LIN {X 0,Y 582.697,Z 999.252,A -85,B 0,C 180,E1 27417.863,E2 27417.863} C_VEL
LIN {X 0,Y 579.637,Z 1018.476,A -85,B 0,C 180,E1 27415.72,E2 27415.72} C_VEL
LIN {X 0,Y 576.832,Z 1036.876,A -85,B 0,C 180,E1 27413.377,E2 27413.377} C_VEL
LIN {X 0,Y 574.399,Z 1053.777,A -85,B 0,C 180,E1 27410.931,E2 27410.931} C_VEL
LIN {X 0,Y 572.425,Z 1069.156,A -85,B 0,C 180,E1 27408.385,E2 27408.385} C_VEL
LIN {X 0,Y 570.966,Z 1081.996,A -85,B 0,C 180,E1 27405.955,E2 27405.955} C_VEL
LIN {X 0,Y 569.794,Z 1094.009,A -85,B 0,C 180,E1 27403.325,E2 27403.325} C_VEL
LIN {X 0,Y 568.899,Z 1104.701,A -85,B 0,C 180,E1 27400.565,E2 27400.565} C_VEL
LIN {X 0,Y 568.443,Z 1112.638,A -85,B 0,C 180,E1 27398.127,E2 27398.127} C_VEL
LIN {X 0,Y 568.122,Z 1119.365,A -85,B 0,C 180,E1 27395.6,E2 27395.6} C_VEL
LIN {X 0,Y 567.953,Z 1124.698,A -85,B 0,C 180,E1 27393.071,E2 27393.071} C_VEL
LIN {X 0,Y 567.932,Z 1128.442,A -85,B 0,C 180,E1 27390.581,E2 27390.581} C_VEL
LIN {X 0,Y 567.917,Z 1130.903,A -85,B 0,C 180,E1 27388.04,E2 27388.04} C_VEL
LIN {X 0,Y 567.902,Z 1131.896,A -85,B 0,C 180,E1 27385.554,E2 27385.554} C_VEL
LIN {X 0,Y 567.866,Z 1131.496,A -85,B 0,C 180,E1 27382.901,E2 27382.901} C_VEL
LIN {X 0,Y 567.918,Z 1129.69,A -85,B 0,C 180,E1 27380.402,E2 27380.402} C_VEL
LIN {X 0,Y 567.966,Z 1126.174,A -85,B 0,C 180,E1 27377.732,E2 27377.732} C_VEL
LIN {X 0,Y 568.103,Z 1120.964,A -85,B 0,C 180,E1 27374.995,E2 27374.995} C_VEL
LIN {X 0,Y 568.345,Z 1114.143,A -85,B 0,C 180,E1 27372.291,E2 27372.291} C_VEL
LIN {X 0,Y 568.803,Z 1106.34,A -85,B 0,C 180,E1 27369.818,E2 27369.818} C_VEL
LIN {X 0,Y 569.536,Z 1096.854,A -85,B 0,C 180,E1 27367.262,E2 27367.262} C_VEL
LIN {X 0,Y 570.678,Z 1084.618,A -85,B 0,C 180,E1 27364.488,E2 27364.488} C_VEL
LIN {X 0,Y 572.097,Z 1071.819,A -85,B 0,C 180,E1 27362.003,E2 27362.003} C_VEL
LIN {X 0,Y 573.974,Z 1057.101,A -85,B 0,C 180,E1 27359.501,E2 27359.501} C_VEL
LIN {X 0,Y 576.32,Z 1040.394,A -85,B 0,C 180,E1 27357.016,E2 27357.016} C_VEL
LIN {X 0,Y 578.934,Z 1023.074,A -85,B 0,C 180,E1 27354.748,E2 27354.748} C_VEL
LIN {X 0,Y 582,Z 1003.502,A -85,B 0,C 180,E1 27352.497,E2 27352.497} C_VEL
LIN {X 0,Y 585.241,Z 983.342,A -85,B 0,C 180,E1 27350.461,E2 27350.461} C_VEL
LIN {X 0,Y 588.632,Z 962.34,A -85,B 0,C 180,E1 27348.586,E2 27348.586} C_VEL
LIN {X 0,Y 592.216,Z 939.835,A -85,B 0,C 180,E1 27346.825,E2 27346.825} C_VEL
LIN {X 0,Y 595.837,Z 916.143,A -85,B 0,C 180,E1 27345.222,E2 27345.222} C_VEL
LIN {X 0,Y 599.193,Z 893.145,A -85,B 0,C 180,E1 27343.868,E2 27343.868} C_VEL
LIN {X 0,Y 602.06,Z 871.003,A -85,B 0,C 180,E1 27342.755,E2 27342.755} C_VEL
LIN {X 0,Y 604.46,Z 849.4,A -85,B 0,C 180,E1 27341.831,E2 27341.831} C_VEL
LIN {X 0,Y 606.973,Z 822.591,A -85,B 0,C 180,E1 27340.888,E2 27340.888} C_VEL
LIN {X 0,Y 608.639,Z 799.863,A -85,B 0,C 180,E1 27340.257,E2 27340.257} C_VEL
LIN {X 0,Y 609.845,Z 778.887,A -85,B 0,C 180,E1 27339.791,E2 27339.791} C_VEL
LIN {X 0,Y 610.75,Z 757.121,A -85,B 0,C 180,E1 27339.422,E2 27339.422} C_VEL
LIN {X 0,Y 615.009,Z 585.018,A -85,B 0,C 180,E1 27337.044,E2 27337.044} C_VEL
LIN {X 0,Y 619.202,Z 468.417,A -85,B 0,C 180,E1 27335.305,E2 27335.305} C_VEL
LIN {X 0,Y 621.386,Z 419.773,A -85,B 0,C 180,E1 27334.516,E2 27334.516} C_VEL
LIN {X 0,Y 613.039,Z 405.628,A -85,B 0,C 180,E1 27332.992,E2 27332.992} C_VEL
LIN {X 0,Y 608.359,Z 397.704,A -85,B 0,C 180,E1 27331.887,E2 27331.887} C_VEL
LIN {X 0,Y 605.73,Z 393.264,A -85,B 0,C 180,E1 27331.075,E2 27331.075} C_VEL
LIN {X 0,Y 603.613,Z 389.51,A -85,B 0,C 180,E1 27330.201,E2 27330.201} C_VEL
LIN {X 0,Y 602.051,Z 387.195,A -85,B 0,C 180,E1 27329.068,E2 27329.068} C_VEL
LIN {X 0,Y 601.397,Z 389.334,A -85,B 0,C 180,E1 27328.306,E2 27328.306} C_VEL
LIN {X 0,Y 601.328,Z 391.857,A -85,B 0,C 180,E1 27327.678,E2 27327.678} C_VEL
LIN {X 0,Y 602.239,Z 397.51,A -85,B 0,C 180,E1 27326.663,E2 27326.663} C_VEL
LIN {X 0,Y 604.241,Z 405.255,A -85,B 0,C 180,E1 27325.619,E2 27325.619} C_VEL
LIN {X 0,Y 608.329,Z 418.436,A -85,B 0,C 180,E1 27324.303,E2 27324.303} C_VEL
LIN {X 0,Y 613.755,Z 430.748,A -85,B 0,C 180,E1 27323.141,E2 27323.141} C_VEL
LIN {X 0,Y 617.349,Z 460.837,A -85,B 0,C 180,E1 27321.984,E2 27321.984} C_VEL
LIN {X 0,Y 619.834,Z 475.835,A -85,B 0,C 180,E1 27321.397,E2 27321.397} C_VEL
LIN {X 0,Y 615.945,Z 588.673,A -85,B 0,C 180,E1 27319.681,E2 27319.681} C_VEL
LIN {X 0,Y 612.665,Z 730.462,A -85,B 0,C 180,E1 27317.702,E2 27317.702} C_VEL
LIN {X 0,Y 609.681,Z 897.665,A -85,B 0,C 180,E1 27315.502,E2 27315.502} C_VEL
LIN {X 0,Y 608.295,Z 927.071,A -85,B 0,C 180,E1 27314.989,E2 27314.989} C_VEL
LIN {X 0,Y 606.632,Z 952.665,A -85,B 0,C 180,E1 27314.385,E2 27314.385} C_VEL
LIN {X 0,Y 605.035,Z 974.265,A -85,B 0,C 180,E1 27313.764,E2 27313.764} C_VEL
LIN {X 0,Y 603.312,Z 995.06,A -85,B 0,C 180,E1 27313.064,E2 27313.064} C_VEL
LIN {X 0,Y 601.59,Z 1014.742,A -85,B 0,C 180,E1 27312.3,E2 27312.3} C_VEL
LIN {X 0,Y 599.545,Z 1035.386,A -85,B 0,C 180,E1 27311.395,E2 27311.395} C_VEL
LIN {X 0,Y 597.906,Z 1050.557,A -85,B 0,C 180,E1 27310.644,E2 27310.644} C_VEL
LIN {X 0,Y 595.718,Z 1066.737,A -85,B 0,C 180,E1 27309.691,E2 27309.691} C_VEL
LIN {X 0,Y 592.722,Z 1086.305,A -85,B 0,C 180,E1 27308.374,E2 27308.374} C_VEL
LIN {X 0,Y 589.851,Z 1104.551,A -85,B 0,C 180,E1 27306.997,E2 27306.997} C_VEL
LIN {X 0,Y 586.954,Z 1122.563,A -85,B 0,C 180,E1 27305.483,E2 27305.483} C_VEL
LIN {X 0,Y 583.573,Z 1143.707,A -85,B 0,C 180,E1 27303.484,E2 27303.484} C_VEL
LIN {X 0,Y 580.57,Z 1162.442,A -85,B 0,C 180,E1 27301.455,E2 27301.455} C_VEL
LIN {X 0,Y 578.226,Z 1177.518,A -85,B 0,C 180,E1 27299.64,E2 27299.64} C_VEL
LIN {X 0,Y 575.845,Z 1193.458,A -85,B 0,C 180,E1 27297.508,E2 27297.508} C_VEL
LIN {X 0,Y 573.558,Z 1210.189,A -85,B 0,C 180,E1 27294.953,E2 27294.953} C_VEL
LIN {X 0,Y 571.964,Z 1222.995,A -85,B 0,C 180,E1 27292.727,E2 27292.727} C_VEL
LIN {X 0,Y 570.657,Z 1234.974,A -85,B 0,C 180,E1 27290.378,E2 27290.378} C_VEL
LIN {X 0,Y 569.454,Z 1247.679,A -85,B 0,C 180,E1 27287.473,E2 27287.473} C_VEL
LIN {X 0,Y 568.84,Z 1256.157,A -85,B 0,C 180,E1 27285.183,E2 27285.183} C_VEL
LIN {X 0,Y 568.409,Z 1263.353,A -85,B 0,C 180,E1 27282.909,E2 27282.909} C_VEL
LIN {X 0,Y 568.135,Z 1269.834,A -85,B 0,C 180,E1 27280.444,E2 27280.444} C_VEL
LIN {X 0,Y 567.953,Z 1275.42,A -85,B 0,C 180,E1 27277.689,E2 27277.689} C_VEL
LIN {X 0,Y 567.923,Z 1278.879,A -85,B 0,C 180,E1 27275.253,E2 27275.253} C_VEL
LIN {X 0,Y 567.91,Z 1280.879,A -85,B 0,C 180,E1 27273.028,E2 27273.028} C_VEL
LIN {X 0,Y 567.875,Z 1281.781,A -85,B 0,C 180,E1 27271.009,E2 27271.009} C_VEL
LIN {X 0,Y 567.875,Z 1281.781,A -85,B 0,C 180,E1 27268.991,E2 27268.991} C_VEL
LIN {X 0,Y 567.91,Z 1280.879,A -85,B 0,C 180,E1 27266.972,E2 27266.972} C_VEL
LIN {X 0,Y 567.923,Z 1278.878,A -85,B 0,C 180,E1 27264.747,E2 27264.747} C_VEL
LIN {X 0,Y 567.955,Z 1275.25,A -85,B 0,C 180,E1 27262.209,E2 27262.209} C_VEL
LIN {X 0,Y 568.142,Z 1269.581,A -85,B 0,C 180,E1 27259.454,E2 27259.454} C_VEL
LIN {X 0,Y 568.418,Z 1263.206,A -85,B 0,C 180,E1 27257.042,E2 27257.042} C_VEL
LIN {X 0,Y 568.843,Z 1256.097,A -85,B 0,C 180,E1 27254.8,E2 27254.8} C_VEL
LIN {X 0,Y 569.489,Z 1247.324,A -85,B 0,C 180,E1 27252.437,E2 27252.437} C_VEL
LIN {X 0,Y 570.67,Z 1234.842,A -85,B 0,C 180,E1 27249.594,E2 27249.594} C_VEL
LIN {X 0,Y 571.965,Z 1222.998,A -85,B 0,C 180,E1 27247.273,E2 27247.273} C_VEL
LIN {X 0,Y 573.468,Z 1210.823,A -85,B 0,C 180,E1 27245.153,E2 27245.153} C_VEL
LIN {X 0,Y 575.643,Z 1195,A -85,B 0,C 180,E1 27242.706,E2 27242.706} C_VEL
LIN {X 0,Y 578.108,Z 1178.291,A -85,B 0,C 180,E1 27240.457,E2 27240.457} C_VEL
LIN {X 0,Y 580.47,Z 1163.078,A -85,B 0,C 180,E1 27238.618,E2 27238.618} C_VEL
LIN {X 0,Y 583.111,Z 1146.446,A -85,B 0,C 180,E1 27236.804,E2 27236.804} C_VEL
LIN {X 0,Y 586.711,Z 1124.077,A -85,B 0,C 180,E1 27234.649,E2 27234.649} C_VEL
LIN {X 0,Y 589.739,Z 1105.21,A -85,B 0,C 180,E1 27233.056,E2 27233.056} C_VEL
LIN {X 0,Y 592.588,Z 1087.11,A -85,B 0,C 180,E1 27231.685,E2 27231.685} C_VEL
LIN {X 0,Y 595.584,Z 1067.54,A -85,B 0,C 180,E1 27230.361,E2 27230.361} C_VEL
LIN {X 0,Y 597.784,Z 1051.537,A -85,B 0,C 180,E1 27229.409,E2 27229.409} C_VEL
LIN {X 0,Y 600.834,Z 1026.776,A -85,B 0,C 180,E1 27228.139,E2 27228.139} C_VEL
LIN {X 0,Y 603.688,Z 1000.444,A -85,B 0,C 180,E1 27227.002,E2 27227.002} C_VEL
LIN {X 0,Y 605.821,Z 979.05,A -85,B 0,C 180,E1 27226.215,E2 27226.215} C_VEL
LIN {X 0,Y 607.671,Z 958.224,A -85,B 0,C 180,E1 27225.563,E2 27225.563} C_VEL
LIN {X 0,Y 609.319,Z 937.399,A -85,B 0,C 180,E1 27225.021,E2 27225.021} C_VEL
LIN {X 0,Y 610.717,Z 916.154,A -85,B 0,C 180,E1 27224.574,E2 27224.574} C_VEL
LIN {X 0,Y 611.99,Z 889.237,A -85,B 0,C 180,E1 27224.137,E2 27224.137} C_VEL
LIN {X 0,Y 616.925,Z 699.679,A -85,B 0,C 180,E1 27221.5,E2 27221.5} C_VEL
LIN {X 0,Y 622.548,Z 518.331,A -85,B 0,C 180,E1 27218.879,E2 27218.879} C_VEL
LIN {X 0,Y 623.894,Z 475.095,A -85,B 0,C 180,E1 27218.216,E2 27218.216} C_VEL
LIN {X 0,Y 616.497,Z 434.81,A -85,B 0,C 180,E1 27216.587,E2 27216.587} C_VEL
LIN {X 0,Y 604.171,Z 415.814,A -85,B 0,C 180,E1 27214.645,E2 27214.645} C_VEL
LIN {X 0,Y 595.164,Z 397.773,A -85,B 0,C 180,E1 27211.952,E2 27211.952} C_VEL
LIN {X 0,Y 587.795,Z 383.94,A -85,B 0,C 180,E1 27209.671,E2 27209.671} C_VEL
LIN {X 0,Y 582.452,Z 374.232,A -85,B 0,C 180,E1 27207.947,E2 27207.947} C_VEL
LIN {X 0,Y 579.549,Z 369.097,A -85,B 0,C 180,E1 27206.985,E2 27206.985} C_VEL
LIN {X 0,Y 577.313,Z 364.965,A -85,B 0,C 180,E1 27206.21,E2 27206.21} C_VEL
LIN {X 0,Y 574.545,Z 360.036,A -85,B 0,C 180,E1 27205.238,E2 27205.238} C_VEL
LIN {X 0,Y 572.463,Z 356.353,A -85,B 0,C 180,E1 27204.496,E2 27204.496} C_VEL
LIN {X 0,Y 569.642,Z 351.574,A -85,B 0,C 180,E1 27203.482,E2 27203.482} C_VEL
LIN {X 0,Y 569.398,Z 350.47,A -85,B 0,C 180,E1 27203.214,E2 27203.214} C_VEL
LIN {X 0,Y 569.361,Z 350.303,A -85,B 0,C 180,E1 27200.026,E2 27200.026} C_VEL
LIN {X 0,Y 569.372,Z 350.311,A -85,B 0,C 180,E1 27196.634,E2 27196.634} C_VEL
LIN {X 0,Y 569.381,Z 350.308,A -85,B 0,C 180,E1 27193.3,E2 27193.3} C_VEL
LIN {X 0,Y 569.352,Z 350.309,A -85,B 0,C 180,E1 27190.013,E2 27190.013} C_VEL
LIN {X 0,Y 569.378,Z 350.31,A -85,B 0,C 180,E1 27186.757,E2 27186.757} C_VEL
LIN {X 0,Y 569.352,Z 350.309,A -85,B 0,C 180,E1 27183.524,E2 27183.524} C_VEL
LIN {X 0,Y 569.366,Z 350.309,A -85,B 0,C 180,E1 27180.101,E2 27180.101} C_VEL
LIN {X 0,Y 569.378,Z 350.302,A -85,B 0,C 180,E1 27176.778,E2 27176.778} C_VEL
LIN {X 0,Y 569.343,Z 350.306,A -85,B 0,C 180,E1 27173.546,E2 27173.546} C_VEL
LIN {X 0,Y 569.382,Z 350.307,A -85,B 0,C 180,E1 27170.294,E2 27170.294} C_VEL
LIN {X 0,Y 569.346,Z 350.307,A -85,B 0,C 180,E1 27167.009,E2 27167.009} C_VEL
LIN {X 0,Y 569.364,Z 350.303,A -85,B 0,C 180,E1 27163.681,E2 27163.681} C_VEL
LIN {X 0,Y 569.372,Z 350.305,A -85,B 0,C 180,E1 27160.402,E2 27160.402} C_VEL
LIN {X 0,Y 569.34,Z 350.301,A -85,B 0,C 180,E1 27157.162,E2 27157.162} C_VEL
LIN {X 0,Y 569.382,Z 350.301,A -85,B 0,C 180,E1 27153.958,E2 27153.958} C_VEL
LIN {X 0,Y 569.333,Z 350.3,A -85,B 0,C 180,E1 27150.775,E2 27150.775} C_VEL
LIN {X 0,Y 569.383,Z 350.3,A -85,B 0,C 180,E1 27147.615,E2 27147.615} C_VEL
LIN {X 0,Y 569.331,Z 350.301,A -85,B 0,C 180,E1 27144.403,E2 27144.403} C_VEL
LIN {X 0,Y 569.362,Z 350.3,A -85,B 0,C 180,E1 27141.075,E2 27141.075} C_VEL
LIN {X 0,Y 569.34,Z 350.3,A -85,B 0,C 180,E1 27137.977,E2 27137.977} C_VEL
LIN {X 0,Y 569.337,Z 350.303,A -85,B 0,C 180,E1 27134.627,E2 27134.627} C_VEL
LIN {X 0,Y 569.367,Z 350.298,A -85,B 0,C 180,E1 27131.457,E2 27131.457} C_VEL
LIN {X 0,Y 569.325,Z 350.305,A -85,B 0,C 180,E1 27128.274,E2 27128.274} C_VEL
LIN {X 0,Y 569.379,Z 350.297,A -85,B 0,C 180,E1 27125.08,E2 27125.08} C_VEL
LIN {X 0,Y 569.318,Z 350.306,A -85,B 0,C 180,E1 27121.913,E2 27121.913} C_VEL
LIN {X 0,Y 569.388,Z 350.296,A -85,B 0,C 180,E1 27118.761,E2 27118.761} C_VEL
LIN {X 0,Y 569.315,Z 350.308,A -85,B 0,C 180,E1 27115.597,E2 27115.597} C_VEL
LIN {X 0,Y 569.372,Z 350.304,A -85,B 0,C 180,E1 27112.4,E2 27112.4} C_VEL
LIN {X 0,Y 569.314,Z 350.312,A -85,B 0,C 180,E1 27109.28,E2 27109.28} C_VEL
LIN {X 0,Y 569.342,Z 350.308,A -85,B 0,C 180,E1 27106.005,E2 27106.005} C_VEL
LIN {X 0,Y 569.337,Z 350.302,A -85,B 0,C 180,E1 27104.779,E2 27104.779} C_VEL
LIN {X 0,Y 568.392,Z 350.431,A -85,B 0,C 180,E1 27104.004,E2 27104.004} C_VEL
LIN {X 0,Y 561.909,Z 351.238,A -85,B 0,C 180,E1 27101.827,E2 27101.827} C_VEL
LIN {X 0,Y 561.367,Z 351.305,A -85,B 0,C 180,E1 27101.26,E2 27101.26} C_VEL
LIN {X 0,Y 561.43,Z 351.293,A -85,B 0,C 180,E1 27098.018,E2 27098.018} C_VEL
LIN {X 0,Y 561.362,Z 351.295,A -85,B 0,C 180,E1 27094.905,E2 27094.905} C_VEL
LIN {X 0,Y 561.401,Z 351.301,A -85,B 0,C 180,E1 27091.633,E2 27091.633} C_VEL
LIN {X 0,Y 561.357,Z 351.297,A -85,B 0,C 180,E1 27088.775,E2 27088.775} C_VEL
LIN {X 0,Y 561.407,Z 351.318,A -85,B 0,C 180,E1 27085.505,E2 27085.505} C_VEL
LIN {X 0,Y 561.492,Z 352.006,A -85,B 0,C 180,E1 27085.199,E2 27085.199} C_VEL
LIN {X 0,Y 563.171,Z 355.462,A -85,B 0,C 180,E1 27084.778,E2 27084.778} C_VEL
LIN {X 0,Y 566.291,Z 358.07,A -85,B 0,C 180,E1 27084.198,E2 27084.198} C_VEL
LIN {X 0,Y 568.698,Z 361.839,A -85,B 0,C 180,E1 27083.717,E2 27083.717} C_VEL
LIN {X 0,Y 571.047,Z 364.138,A -85,B 0,C 180,E1 27083.291,E2 27083.291} C_VEL
LIN {X 0,Y 574.102,Z 368.286,A -85,B 0,C 180,E1 27082.721,E2 27082.721} C_VEL
LIN {X 0,Y 575.942,Z 370.323,A -85,B 0,C 180,E1 27082.396,E2 27082.396} C_VEL
LIN {X 0,Y 579.512,Z 374.773,A -85,B 0,C 180,E1 27081.767,E2 27081.767} C_VEL
LIN {X 0,Y 586.209,Z 383.24,A -85,B 0,C 180,E1 27080.625,E2 27080.625} C_VEL
LIN {X 0,Y 594.382,Z 393.676,A -85,B 0,C 180,E1 27079.292,E2 27079.292} C_VEL
LIN {X 0,Y 604.893,Z 407.519,A -85,B 0,C 180,E1 27077.669,E2 27077.669} C_VEL
LIN {X 0,Y 616.339,Z 423.555,A -85,B 0,C 180,E1 27076.012,E2 27076.012} C_VEL
LIN {X 0,Y 616.87,Z 424.779,A -85,B 0,C 180,E1 27075.929,E2 27075.929} C_VEL
LIN {X 0,Y 610.091,Z 626.628,A -85,B 0,C 180,E1 27072.993,E2 27072.993} C_VEL
LIN {X 0,Y 606.036,Z 760.175,A -85,B 0,C 180,E1 27071.091,E2 27071.091} C_VEL
LIN {X 0,Y 604.393,Z 788.186,A -85,B 0,C 180,E1 27070.545,E2 27070.545} C_VEL
LIN {X 0,Y 602.314,Z 813.584,A -85,B 0,C 180,E1 27069.87,E2 27069.87} C_VEL
LIN {X 0,Y 600.068,Z 836.778,A -85,B 0,C 180,E1 27069.11,E2 27069.11} C_VEL
LIN {X 0,Y 597.067,Z 863.226,A -85,B 0,C 180,E1 27068.049,E2 27068.049} C_VEL
LIN {X 0,Y 593.907,Z 886.824,A -85,B 0,C 180,E1 27066.904,E2 27066.904} C_VEL
LIN {X 0,Y 590.552,Z 909.945,A -85,B 0,C 180,E1 27065.599,E2 27065.599} C_VEL
LIN {X 0,Y 586.909,Z 932.754,A -85,B 0,C 180,E1 27064.097,E2 27064.097} C_VEL
LIN {X 0,Y 583.066,Z 955.615,A -85,B 0,C 180,E1 27062.363,E2 27062.363} C_VEL
LIN {X 0,Y 579.224,Z 978.099,A -85,B 0,C 180,E1 27060.416,E2 27060.416} C_VEL
LIN {X 0,Y 575.746,Z 998.788,A -85,B 0,C 180,E1 27058.367,E2 27058.367} C_VEL
LIN {X 0,Y 572.554,Z 1017.785,A -85,B 0,C 180,E1 27056.23,E2 27056.23} C_VEL
LIN {X 0,Y 569.57,Z 1035.993,A -85,B 0,C 180,E1 27053.899,E2 27053.899} C_VEL
LIN {X 0,Y 566.943,Z 1053.353,A -85,B 0,C 180,E1 27051.368,E2 27051.368} C_VEL
LIN {X 0,Y 564.825,Z 1068.753,A -85,B 0,C 180,E1 27048.796,E2 27048.796} C_VEL
LIN {X 0,Y 563.216,Z 1081.959,A -85,B 0,C 180,E1 27046.266,E2 27046.266} C_VEL
LIN {X 0,Y 561.946,Z 1093.973,A -85,B 0,C 180,E1 27043.6,E2 27043.6} C_VEL
LIN {X 0,Y 561,Z 1104.49,A -85,B 0,C 180,E1 27040.853,E2 27040.853} C_VEL
LIN {X 0,Y 560.508,Z 1112.474,A -85,B 0,C 180,E1 27038.375,E2 27038.375} C_VEL
LIN {X 0,Y 560.143,Z 1119.165,A -85,B 0,C 180,E1 27035.839,E2 27035.839} C_VEL
LIN {X 0,Y 559.976,Z 1124.458,A -85,B 0,C 180,E1 27033.317,E2 27033.317} C_VEL
LIN {X 0,Y 559.938,Z 1128.378,A -85,B 0,C 180,E1 27030.712,E2 27030.712} C_VEL
LIN {X 0,Y 559.919,Z 1130.897,A -85,B 0,C 180,E1 27028.096,E2 27028.096} C_VEL
LIN {X 0,Y 559.903,Z 1131.889,A -85,B 0,C 180,E1 27025.601,E2 27025.601} C_VEL
LIN {X 0,Y 559.866,Z 1131.517,A -85,B 0,C 180,E1 27022.913,E2 27022.913} C_VEL
LIN {X 0,Y 559.918,Z 1129.714,A -85,B 0,C 180,E1 27020.361,E2 27020.361} C_VEL
LIN {X 0,Y 559.97,Z 1126.24,A -85,B 0,C 180,E1 27017.671,E2 27017.671} C_VEL
LIN {X 0,Y 560.115,Z 1121.065,A -85,B 0,C 180,E1 27014.896,E2 27014.896} C_VEL
LIN {X 0,Y 560.39,Z 1114.136,A -85,B 0,C 180,E1 27012.105,E2 27012.105} C_VEL
LIN {X 0,Y 560.859,Z 1106.5,A -85,B 0,C 180,E1 27009.646,E2 27009.646} C_VEL
LIN {X 0,Y 561.655,Z 1097.056,A -85,B 0,C 180,E1 27007.056,E2 27007.056} C_VEL
LIN {X 0,Y 562.851,Z 1085.036,A -85,B 0,C 180,E1 27004.279,E2 27004.279} C_VEL
LIN {X 0,Y 564.374,Z 1072.104,A -85,B 0,C 180,E1 27001.726,E2 27001.726} C_VEL
LIN {X 0,Y 566.359,Z 1057.44,A -85,B 0,C 180,E1 26999.191,E2 26999.191} C_VEL
LIN {X 0,Y 568.856,Z 1040.789,A -85,B 0,C 180,E1 26996.675,E2 26996.675} C_VEL
LIN {X 0,Y 571.609,Z 1023.509,A -85,B 0,C 180,E1 26994.378,E2 26994.378} C_VEL
LIN {X 0,Y 574.696,Z 1004.869,A -85,B 0,C 180,E1 26992.2,E2 26992.2} C_VEL
LIN {X 0,Y 578.179,Z 984.393,A -85,B 0,C 180,E1 26990.092,E2 26990.092} C_VEL
LIN {X 0,Y 581.647,Z 964.115,A -85,B 0,C 180,E1 26988.246,E2 26988.246} C_VEL
LIN {X 0,Y 585.484,Z 941.12,A -85,B 0,C 180,E1 26986.419,E2 26986.419} C_VEL
LIN {X 0,Y 588.983,Z 920.111,A -85,B 0,C 180,E1 26984.945,E2 26984.945} C_VEL
LIN {X 0,Y 592.579,Z 896.742,A -85,B 0,C 180,E1 26983.532,E2 26983.532} C_VEL
LIN {X 0,Y 595.368,Z 875.755,A -85,B 0,C 180,E1 26982.455,E2 26982.455} C_VEL
LIN {X 0,Y 597.7,Z 855.684,A -85,B 0,C 180,E1 26981.568,E2 26981.568} C_VEL
LIN {X 0,Y 599.695,Z 835.977,A -85,B 0,C 180,E1 26980.824,E2 26980.824} C_VEL
LIN {X 0,Y 601.598,Z 813.781,A -85,B 0,C 180,E1 26980.123,E2 26980.123} C_VEL
LIN {X 0,Y 603.385,Z 785.822,A -85,B 0,C 180,E1 26979.435,E2 26979.435} C_VEL
LIN {X 0,Y 604.388,Z 763.833,A -85,B 0,C 180,E1 26979.037,E2 26979.037} C_VEL
LIN {X 0,Y 609.063,Z 593.316,A -85,B 0,C 180,E1 26976.634,E2 26976.634} C_VEL
LIN {X 0,Y 613.387,Z 483.426,A -85,B 0,C 180,E1 26974.965,E2 26974.965} C_VEL
LIN {X 0,Y 616.514,Z 424.015,A -85,B 0,C 180,E1 26973.988,E2 26973.988} C_VEL
LIN {X 0,Y 609.78,Z 411.938,A -85,B 0,C 180,E1 26972.64,E2 26972.64} C_VEL
LIN {X 0,Y 605.672,Z 404.517,A -85,B 0,C 180,E1 26971.576,E2 26971.576} C_VEL
LIN {X 0,Y 603.262,Z 400.207,A -85,B 0,C 180,E1 26970.758,E2 26970.758} C_VEL
LIN {X 0,Y 601.745,Z 397.053,A -85,B 0,C 180,E1 26969.989,E2 26969.989} C_VEL
LIN {X 0,Y 600.517,Z 395.257,A -85,B 0,C 180,E1 26969.035,E2 26969.035} C_VEL
LIN {X 0,Y 599.795,Z 398.364,A -85,B 0,C 180,E1 26968.127,E2 26968.127} C_VEL
LIN {X 0,Y 599.984,Z 403.477,A -85,B 0,C 180,E1 26967.149,E2 26967.149} C_VEL
LIN {X 0,Y 601.398,Z 410.908,A -85,B 0,C 180,E1 26966.096,E2 26966.096} C_VEL
LIN {X 0,Y 603.673,Z 420.099,A -85,B 0,C 180,E1 26965.12,E2 26965.12} C_VEL
LIN {X 0,Y 608.28,Z 432.666,A -85,B 0,C 180,E1 26963.878,E2 26963.878} C_VEL
LIN {X 0,Y 609.407,Z 435.449,A -85,B 0,C 180,E1 26963.62,E2 26963.62} C_VEL
LIN {X 0,Y 612.454,Z 464.305,A -85,B 0,C 180,E1 26962.478,E2 26962.478} C_VEL
LIN {X 0,Y 614.524,Z 477.977,A -85,B 0,C 180,E1 26961.931,E2 26961.931} C_VEL
LIN {X 0,Y 610.225,Z 586.077,A -85,B 0,C 180,E1 26960.238,E2 26960.238} C_VEL
LIN {X 0,Y 606.925,Z 708.219,A -85,B 0,C 180,E1 26958.483,E2 26958.483} C_VEL
LIN {X 0,Y 603.873,Z 866.055,A -85,B 0,C 180,E1 26956.372,E2 26956.372} C_VEL
LIN {X 0,Y 602.793,Z 905.519,A -85,B 0,C 180,E1 26955.813,E2 26955.813} C_VEL
LIN {X 0,Y 601.337,Z 931.07,A -85,B 0,C 180,E1 26955.319,E2 26955.319} C_VEL
LIN {X 0,Y 599.804,Z 953.328,A -85,B 0,C 180,E1 26954.776,E2 26954.776} C_VEL
LIN {X 0,Y 598.084,Z 975.19,A -85,B 0,C 180,E1 26954.131,E2 26954.131} C_VEL
LIN {X 0,Y 596.035,Z 998.438,A -85,B 0,C 180,E1 26953.323,E2 26953.323} C_VEL
LIN {X 0,Y 593.246,Z 1027.217,A -85,B 0,C 180,E1 26952.129,E2 26952.129} C_VEL
LIN {X 0,Y 590.82,Z 1049.569,A -85,B 0,C 180,E1 26951.043,E2 26951.043} C_VEL
LIN {X 0,Y 588.511,Z 1069.45,A -85,B 0,C 180,E1 26949.957,E2 26949.957} C_VEL
LIN {X 0,Y 586.729,Z 1083.273,A -85,B 0,C 180,E1 26949.09,E2 26949.09} C_VEL
LIN {X 0,Y 583.678,Z 1101.879,A -85,B 0,C 180,E1 26947.702,E2 26947.702} C_VEL
LIN {X 0,Y 580.751,Z 1119.212,A -85,B 0,C 180,E1 26946.256,E2 26946.256} C_VEL
LIN {X 0,Y 577.947,Z 1135.653,A -85,B 0,C 180,E1 26944.736,E2 26944.736} C_VEL
LIN {X 0,Y 575.111,Z 1152.32,A -85,B 0,C 180,E1 26943.028,E2 26943.028} C_VEL
LIN {X 0,Y 571.752,Z 1172.446,A -85,B 0,C 180,E1 26940.707,E2 26940.707} C_VEL
LIN {X 0,Y 569.146,Z 1188.834,A -85,B 0,C 180,E1 26938.545,E2 26938.545} C_VEL
LIN {X 0,Y 567.026,Z 1202.775,A -85,B 0,C 180,E1 26936.496,E2 26936.496} C_VEL
LIN {X 0,Y 564.965,Z 1217.795,A -85,B 0,C 180,E1 26934.02,E2 26934.02} C_VEL
LIN {X 0,Y 563.262,Z 1231.233,A -85,B 0,C 180,E1 26931.449,E2 26931.449} C_VEL
LIN {X 0,Y 562.198,Z 1241.065,A -85,B 0,C 180,E1 26929.317,E2 26929.317} C_VEL
LIN {X 0,Y 561.358,Z 1250.109,A -85,B 0,C 180,E1 26927.091,E2 26927.091} C_VEL
LIN {X 0,Y 560.696,Z 1258.98,A -85,B 0,C 180,E1 26924.563,E2 26924.563} C_VEL
LIN {X 0,Y 560.263,Z 1267.037,A -85,B 0,C 180,E1 26921.739,E2 26921.739} C_VEL
LIN {X 0,Y 560.02,Z 1272.297,A -85,B 0,C 180,E1 26919.454,E2 26919.454} C_VEL
LIN {X 0,Y 559.966,Z 1276.375,A -85,B 0,C 180,E1 26917.18,E2 26917.18} C_VEL
LIN {X 0,Y 559.92,Z 1279.444,A -85,B 0,C 180,E1 26914.814,E2 26914.814} C_VEL
LIN {X 0,Y 559.911,Z 1281.549,A -85,B 0,C 180,E1 26912.047,E2 26912.047} C_VEL
LIN {X 0,Y 559.865,Z 1281.872,A -85,B 0,C 180,E1 26909.386,E2 26909.386} C_VEL
LIN {X 0,Y 559.908,Z 1281.083,A -85,B 0,C 180,E1 26907.236,E2 26907.236} C_VEL
LIN {X 0,Y 559.922,Z 1279.216,A -85,B 0,C 180,E1 26904.98,E2 26904.98} C_VEL
LIN {X 0,Y 559.964,Z 1276.214,A -85,B 0,C 180,E1 26902.717,E2 26902.717} C_VEL
LIN {X 0,Y 560.05,Z 1271.677,A -85,B 0,C 180,E1 26900.235,E2 26900.235} C_VEL
LIN {X 0,Y 560.377,Z 1264.563,A -85,B 0,C 180,E1 26897.322,E2 26897.322} C_VEL
LIN {X 0,Y 560.865,Z 1256.86,A -85,B 0,C 180,E1 26894.807,E2 26894.807} C_VEL
LIN {X 0,Y 561.464,Z 1248.894,A -85,B 0,C 180,E1 26892.592,E2 26892.592} C_VEL
LIN {X 0,Y 562.463,Z 1238.768,A -85,B 0,C 180,E1 26890.151,E2 26890.151} C_VEL
LIN {X 0,Y 563.985,Z 1225.29,A -85,B 0,C 180,E1 26887.374,E2 26887.374} C_VEL
LIN {X 0,Y 565.604,Z 1212.727,A -85,B 0,C 180,E1 26885.119,E2 26885.119} C_VEL
LIN {X 0,Y 567.451,Z 1199.973,A -85,B 0,C 180,E1 26883.074,E2 26883.074} C_VEL
LIN {X 0,Y 570.049,Z 1183.16,A -85,B 0,C 180,E1 26880.664,E2 26880.664} C_VEL
LIN {X 0,Y 572.959,Z 1165.217,A -85,B 0,C 180,E1 26878.431,E2 26878.431} C_VEL
LIN {X 0,Y 575.567,Z 1149.573,A -85,B 0,C 180,E1 26876.679,E2 26876.679} C_VEL
LIN {X 0,Y 578.358,Z 1133.26,A -85,B 0,C 180,E1 26875.032,E2 26875.032} C_VEL
LIN {X 0,Y 581.907,Z 1112.512,A -85,B 0,C 180,E1 26873.153,E2 26873.153} C_VEL
LIN {X 0,Y 585.626,Z 1089.964,A -85,B 0,C 180,E1 26871.388,E2 26871.388} C_VEL
LIN {X 0,Y 587.965,Z 1074.183,A -85,B 0,C 180,E1 26870.315,E2 26870.315} C_VEL
LIN {X 0,Y 590.775,Z 1053.508,A -85,B 0,C 180,E1 26869.081,E2 26869.081} C_VEL
LIN {X 0,Y 593.429,Z 1032.955,A -85,B 0,C 180,E1 26867.993,E2 26867.993} C_VEL
LIN {X 0,Y 596.033,Z 1011.472,A -85,B 0,C 180,E1 26866.993,E2 26866.993} C_VEL
LIN {X 0,Y 599.003,Z 984.545,A -85,B 0,C 180,E1 26865.921,E2 26865.921} C_VEL
LIN {X 0,Y 601.341,Z 959.877,A -85,B 0,C 180,E1 26865.121,E2 26865.121} C_VEL
LIN {X 0,Y 603.115,Z 938.888,A -85,B 0,C 180,E1 26864.56,E2 26864.56} C_VEL
LIN {X 0,Y 604.572,Z 918.293,A -85,B 0,C 180,E1 26864.112,E2 26864.112} C_VEL
LIN {X 0,Y 605.7,Z 897.704,A -85,B 0,C 180,E1 26863.759,E2 26863.759} C_VEL
LIN {X 0,Y 612.052,Z 678.911,A -85,B 0,C 180,E1 26860.656,E2 26860.656} C_VEL
LIN {X 0,Y 618.87,Z 478.003,A -85,B 0,C 180,E1 26857.701,E2 26857.701} C_VEL
LIN {X 0,Y 611.98,Z 439.784,A -85,B 0,C 180,E1 26856.145,E2 26856.145} C_VEL
LIN {X 0,Y 599.705,Z 420.875,A -85,B 0,C 180,E1 26854.186,E2 26854.186} C_VEL
LIN {X 0,Y 594.941,Z 413.617,A -85,B 0,C 180,E1 26853.338,E2 26853.338} C_VEL
LIN {X 0,Y 586.835,Z 397.841,A -85,B 0,C 180,E1 26850.855,E2 26850.855} C_VEL
LIN {X 0,Y 579.958,Z 384.894,A -85,B 0,C 180,E1 26848.639,E2 26848.639} C_VEL
LIN {X 0,Y 574.728,Z 375.435,A -85,B 0,C 180,E1 26846.894,E2 26846.894} C_VEL
LIN {X 0,Y 572.184,Z 370.858,A -85,B 0,C 180,E1 26846.016,E2 26846.016} C_VEL
LIN {X 0,Y 569.334,Z 365.857,A -85,B 0,C 180,E1 26845.013,E2 26845.013} C_VEL
LIN {X 0,Y 566.709,Z 361.14,A -85,B 0,C 180,E1 26844.053,E2 26844.053} C_VEL
LIN {X 0,Y 564.6,Z 357.394,A -85,B 0,C 180,E1 26843.262,E2 26843.262} C_VEL
LIN {X 0,Y 563.477,Z 355.7,A -85,B 0,C 180,E1 26842.868,E2 26842.868} C_VEL
LIN {X 0,Y 561.68,Z 352.556,A -85,B 0,C 180,E1 26842.173,E2 26842.173} C_VEL
LIN {X 0,Y 561.455,Z 351.454,A -85,B 0,C 180,E1 26841.901,E2 26841.901} C_VEL
LIN {X 0,Y 561.422,Z 351.282,A -85,B 0,C 180,E1 26838.483,E2 26838.483} C_VEL
LIN {X 0,Y 561.436,Z 351.279,A -85,B 0,C 180,E1 26835.146,E2 26835.146} C_VEL
LIN {X 0,Y 561.412,Z 351.281,A -85,B 0,C 180,E1 26831.923,E2 26831.923} C_VEL
LIN {X 0,Y 561.44,Z 351.279,A -85,B 0,C 180,E1 26828.604,E2 26828.604} C_VEL
LIN {X 0,Y 561.428,Z 351.278,A -85,B 0,C 180,E1 26825.314,E2 26825.314} C_VEL
LIN {X 0,Y 561.411,Z 351.281,A -85,B 0,C 180,E1 26821.939,E2 26821.939} C_VEL
LIN {X 0,Y 561.442,Z 351.292,A -85,B 0,C 180,E1 26818.673,E2 26818.673} C_VEL
LIN {X 0,Y 561.407,Z 351.294,A -85,B 0,C 180,E1 26815.403,E2 26815.403} C_VEL
LIN {X 0,Y 561.444,Z 351.298,A -85,B 0,C 180,E1 26812.118,E2 26812.118} C_VEL
LIN {X 0,Y 561.423,Z 351.294,A -85,B 0,C 180,E1 26808.806,E2 26808.806} C_VEL
LIN {X 0,Y 561.405,Z 351.297,A -85,B 0,C 180,E1 26805.456,E2 26805.456} C_VEL
LIN {X 0,Y 561.444,Z 351.285,A -85,B 0,C 180,E1 26802.162,E2 26802.162} C_VEL
LIN {X 0,Y 561.399,Z 351.298,A -85,B 0,C 180,E1 26798.913,E2 26798.913} C_VEL
LIN {X 0,Y 561.44,Z 351.29,A -85,B 0,C 180,E1 26795.707,E2 26795.707} C_VEL
LIN {X 0,Y 561.404,Z 351.296,A -85,B 0,C 180,E1 26792.492,E2 26792.492} C_VEL
LIN {X 0,Y 561.404,Z 351.301,A -85,B 0,C 180,E1 26789.021,E2 26789.021} C_VEL
LIN {X 0,Y 561.443,Z 351.294,A -85,B 0,C 180,E1 26785.752,E2 26785.752} C_VEL
LIN {X 0,Y 561.39,Z 351.3,A -85,B 0,C 180,E1 26782.473,E2 26782.473} C_VEL
LIN {X 0,Y 561.451,Z 351.297,A -85,B 0,C 180,E1 26779.321,E2 26779.321} C_VEL
LIN {X 0,Y 561.39,Z 351.299,A -85,B 0,C 180,E1 26776.144,E2 26776.144} C_VEL
LIN {X 0,Y 561.416,Z 351.297,A -85,B 0,C 180,E1 26772.796,E2 26772.796} C_VEL
LIN {X 0,Y 561.395,Z 351.299,A -85,B 0,C 180,E1 26769.747,E2 26769.747} C_VEL
LIN {X 0,Y 561.394,Z 351.296,A -85,B 0,C 180,E1 26766.377,E2 26766.377} C_VEL
LIN {X 0,Y 561.427,Z 351.295,A -85,B 0,C 180,E1 26763.168,E2 26763.168} C_VEL
LIN {X 0,Y 561.378,Z 351.293,A -85,B 0,C 180,E1 26759.915,E2 26759.915} C_VEL
LIN {X 0,Y 561.441,Z 351.286,A -85,B 0,C 180,E1 26756.78,E2 26756.78} C_VEL
LIN {X 0,Y 561.373,Z 351.288,A -85,B 0,C 180,E1 26753.625,E2 26753.625} C_VEL
LIN {X 0,Y 561.437,Z 351.286,A -85,B 0,C 180,E1 26750.43,E2 26750.43} C_VEL
LIN {X 0,Y 561.372,Z 351.297,A -85,B 0,C 180,E1 26747.304,E2 26747.304} C_VEL
LIN {X 0,Y 561.411,Z 351.3,A -85,B 0,C 180,E1 26744.017,E2 26744.017} C_VEL
LIN {X 0,Y 561.367,Z 351.305,A -85,B 0,C 180,E1 26741.26,E2 26741.26} C_VEL
LIN {X 0,Y 560.396,Z 351.424,A -85,B 0,C 180,E1 26740.474,E2 26740.474} C_VEL
LIN {X 0,Y 553.927,Z 352.23,A -85,B 0,C 180,E1 26738.21,E2 26738.21} C_VEL
LIN {X 0,Y 553.452,Z 352.283,A -85,B 0,C 180,E1 26737.692,E2 26737.692} C_VEL
LIN {X 0,Y 553.429,Z 352.283,A -85,B 0,C 180,E1 26734.767,E2 26734.767} C_VEL
LIN {X 0,Y 553.436,Z 352.294,A -85,B 0,C 180,E1 26731.346,E2 26731.346} C_VEL
LIN {X 0,Y 553.431,Z 352.272,A -85,B 0,C 180,E1 26728.447,E2 26728.447} C_VEL
LIN {X 0,Y 553.438,Z 352.435,A -85,B 0,C 180,E1 26726.686,E2 26726.686} C_VEL
LIN {X 0,Y 553.786,Z 353.828,A -85,B 0,C 180,E1 26726.403,E2 26726.403} C_VEL
LIN {X 0,Y 555.798,Z 356.971,A -85,B 0,C 180,E1 26725.951,E2 26725.951} C_VEL
LIN {X 0,Y 558.265,Z 359.047,A -85,B 0,C 180,E1 26725.48,E2 26725.48} C_VEL
LIN {X 0,Y 560.531,Z 362.677,A -85,B 0,C 180,E1 26725.011,E2 26725.011} C_VEL
LIN {X 0,Y 563.446,Z 365.348,A -85,B 0,C 180,E1 26724.468,E2 26724.468} C_VEL
LIN {X 0,Y 566.509,Z 369.479,A -85,B 0,C 180,E1 26723.87,E2 26723.87} C_VEL
LIN {X 0,Y 568.181,Z 371.299,A -85,B 0,C 180,E1 26723.559,E2 26723.559} C_VEL
LIN {X 0,Y 571.755,Z 375.779,A -85,B 0,C 180,E1 26722.893,E2 26722.893} C_VEL
LIN {X 0,Y 583.099,Z 390.078,A -85,B 0,C 180,E1 26720.898,E2 26720.898} C_VEL
LIN {X 0,Y 594.195,Z 404.349,A -85,B 0,C 180,E1 26719.088,E2 26719.088} C_VEL
LIN {X 0,Y 605.476,Z 419.621,A -85,B 0,C 180,E1 26717.356,E2 26717.356} C_VEL
LIN {X 0,Y 611.65,Z 428.622,A -85,B 0,C 180,E1 26716.453,E2 26716.453} C_VEL
LIN {X 0,Y 604.463,Z 631.198,A -85,B 0,C 180,E1 26713.481,E2 26713.481} C_VEL
LIN {X 0,Y 600.297,Z 760.573,A -85,B 0,C 180,E1 26711.62,E2 26711.62} C_VEL
LIN {X 0,Y 598.642,Z 788.234,A -85,B 0,C 180,E1 26711.082,E2 26711.082} C_VEL
LIN {X 0,Y 596.494,Z 813.775,A -85,B 0,C 180,E1 26710.403,E2 26710.403} C_VEL
LIN {X 0,Y 594.337,Z 835.377,A -85,B 0,C 180,E1 26709.697,E2 26709.697} C_VEL
LIN {X 0,Y 591.533,Z 859.691,A -85,B 0,C 180,E1 26708.742,E2 26708.742} C_VEL
LIN {X 0,Y 588.009,Z 885.661,A -85,B 0,C 180,E1 26707.505,E2 26707.505} C_VEL
LIN {X 0,Y 584.657,Z 908.089,A -85,B 0,C 180,E1 26706.25,E2 26706.25} C_VEL
LIN {X 0,Y 580.833,Z 931.382,A -85,B 0,C 180,E1 26704.728,E2 26704.728} C_VEL
LIN {X 0,Y 577.048,Z 952.708,A -85,B 0,C 180,E1 26703.112,E2 26703.112} C_VEL
LIN {X 0,Y 572.973,Z 975.24,A -85,B 0,C 180,E1 26701.168,E2 26701.168} C_VEL
LIN {X 0,Y 569.272,Z 995.884,A -85,B 0,C 180,E1 26699.145,E2 26699.145} C_VEL
LIN {X 0,Y 565.89,Z 1014.764,A -85,B 0,C 180,E1 26697.03,E2 26697.03} C_VEL
LIN {X 0,Y 562.571,Z 1033.962,A -85,B 0,C 180,E1 26694.591,E2 26694.591} C_VEL
LIN {X 0,Y 559.951,Z 1050.311,A -85,B 0,C 180,E1 26692.231,E2 26692.231} C_VEL
LIN {X 0,Y 557.578,Z 1065.924,A -85,B 0,C 180,E1 26689.654,E2 26689.654} C_VEL
LIN {X 0,Y 555.707,Z 1079.861,A -85,B 0,C 180,E1 26687.006,E2 26687.006} C_VEL
LIN {X 0,Y 554.265,Z 1092.371,A -85,B 0,C 180,E1 26684.261,E2 26684.261} C_VEL
LIN {X 0,Y 553.26,Z 1102.923,A -85,B 0,C 180,E1 26681.55,E2 26681.55} C_VEL
LIN {X 0,Y 552.593,Z 1111.946,A -85,B 0,C 180,E1 26678.752,E2 26678.752} C_VEL
LIN {X 0,Y 552.172,Z 1119.038,A -85,B 0,C 180,E1 26676.052,E2 26676.052} C_VEL
LIN {X 0,Y 552.004,Z 1124.275,A -85,B 0,C 180,E1 26673.537,E2 26673.537} C_VEL
LIN {X 0,Y 551.936,Z 1128.333,A -85,B 0,C 180,E1 26670.831,E2 26670.831} C_VEL
LIN {X 0,Y 551.918,Z 1130.85,A -85,B 0,C 180,E1 26668.219,E2 26668.219} C_VEL
LIN {X 0,Y 551.905,Z 1131.881,A -85,B 0,C 180,E1 26665.658,E2 26665.658} C_VEL
LIN {X 0,Y 551.867,Z 1131.538,A -85,B 0,C 180,E1 26662.926,E2 26662.926} C_VEL
LIN {X 0,Y 551.919,Z 1129.764,A -85,B 0,C 180,E1 26660.355,E2 26660.355} C_VEL
LIN {X 0,Y 551.972,Z 1126.306,A -85,B 0,C 180,E1 26657.609,E2 26657.609} C_VEL
LIN {X 0,Y 552.126,Z 1121.166,A -85,B 0,C 180,E1 26654.794,E2 26654.794} C_VEL
LIN {X 0,Y 552.42,Z 1114.403,A -85,B 0,C 180,E1 26652.014,E2 26652.014} C_VEL
LIN {X 0,Y 552.92,Z 1106.67,A -85,B 0,C 180,E1 26649.472,E2 26649.472} C_VEL
LIN {X 0,Y 553.775,Z 1097.255,A -85,B 0,C 180,E1 26646.844,E2 26646.844} C_VEL
LIN {X 0,Y 555.05,Z 1085.271,A -85,B 0,C 180,E1 26644.029,E2 26644.029} C_VEL
LIN {X 0,Y 556.666,Z 1072.39,A -85,B 0,C 180,E1 26641.441,E2 26641.441} C_VEL
LIN {X 0,Y 558.852,Z 1057.15,A -85,B 0,C 180,E1 26638.77,E2 26638.77} C_VEL
LIN {X 0,Y 561.407,Z 1041.186,A -85,B 0,C 180,E1 26636.324,E2 26636.324} C_VEL
LIN {X 0,Y 564.309,Z 1023.938,A -85,B 0,C 180,E1 26633.999,E2 26633.999} C_VEL
LIN {X 0,Y 567.569,Z 1005.347,A -85,B 0,C 180,E1 26631.796,E2 26631.796} C_VEL
LIN {X 0,Y 571.319,Z 984.428,A -85,B 0,C 180,E1 26629.615,E2 26629.615} C_VEL
LIN {X 0,Y 575.168,Z 963.034,A -85,B 0,C 180,E1 26627.653,E2 26627.653} C_VEL
LIN {X 0,Y 579.037,Z 942.335,A -85,B 0,C 180,E1 26625.959,E2 26625.959} C_VEL
LIN {X 0,Y 582.533,Z 921.973,A -85,B 0,C 180,E1 26624.52,E2 26624.52} C_VEL
LIN {X 0,Y 586.232,Z 898.584,A -85,B 0,C 180,E1 26623.094,E2 26623.094} C_VEL
LIN {X 0,Y 589.078,Z 877.478,A -85,B 0,C 180,E1 26622.006,E2 26622.006} C_VEL
LIN {X 0,Y 591.342,Z 858.493,A -85,B 0,C 180,E1 26621.158,E2 26621.158} C_VEL
LIN {X 0,Y 593.383,Z 838.9,A -85,B 0,C 180,E1 26620.407,E2 26620.407} C_VEL
LIN {X 0,Y 595.234,Z 817.839,A -85,B 0,C 180,E1 26619.729,E2 26619.729} C_VEL
LIN {X 0,Y 597.078,Z 791.098,A -85,B 0,C 180,E1 26619.041,E2 26619.041} C_VEL
LIN {X 0,Y 598.188,Z 767.105,A -85,B 0,C 180,E1 26618.589,E2 26618.589} C_VEL
LIN {X 0,Y 603.084,Z 604.353,A -85,B 0,C 180,E1 26616.254,E2 26616.254} C_VEL
LIN {X 0,Y 607.41,Z 503.356,A -85,B 0,C 180,E1 26614.692,E2 26614.692} C_VEL
LIN {X 0,Y 611.779,Z 428.207,A -85,B 0,C 180,E1 26613.433,E2 26613.433} C_VEL
LIN {X 0,Y 606.587,Z 418.193,A -85,B 0,C 180,E1 26612.272,E2 26612.272} C_VEL
LIN {X 0,Y 603.124,Z 411.446,A -85,B 0,C 180,E1 26611.281,E2 26611.281} C_VEL
LIN {X 0,Y 601.042,Z 407.288,A -85,B 0,C 180,E1 26610.464,E2 26610.464} C_VEL
LIN {X 0,Y 599.856,Z 404.578,A -85,B 0,C 180,E1 26609.775,E2 26609.775} C_VEL
LIN {X 0,Y 599.047,Z 403.331,A -85,B 0,C 180,E1 26609.084,E2 26609.084} C_VEL
LIN {X 0,Y 598.228,Z 406.179,A -85,B 0,C 180,E1 26608.292,E2 26608.292} C_VEL
LIN {X 0,Y 598.183,Z 411.288,A -85,B 0,C 180,E1 26607.343,E2 26607.343} C_VEL
LIN {X 0,Y 599.24,Z 419.036,A -85,B 0,C 180,E1 26606.274,E2 26606.274} C_VEL
LIN {X 0,Y 602.321,Z 432.128,A -85,B 0,C 180,E1 26604.925,E2 26604.925} C_VEL
LIN {X 0,Y 605.259,Z 440.21,A -85,B 0,C 180,E1 26604.123,E2 26604.123} C_VEL
LIN {X 0,Y 607.745,Z 467.532,A -85,B 0,C 180,E1 26603.005,E2 26603.005} C_VEL
LIN {X 0,Y 609.394,Z 479.973,A -85,B 0,C 180,E1 26602.486,E2 26602.486} C_VEL
LIN {X 0,Y 604.674,Z 583.936,A -85,B 0,C 180,E1 26600.811,E2 26600.811} C_VEL
LIN {X 0,Y 601.021,Z 698.94,A -85,B 0,C 180,E1 26599.105,E2 26599.105} C_VEL
LIN {X 0,Y 597.908,Z 841.147,A -85,B 0,C 180,E1 26597.157,E2 26597.157} C_VEL
LIN {X 0,Y 596.57,Z 898.996,A -85,B 0,C 180,E1 26596.364,E2 26596.364} C_VEL
LIN {X 0,Y 594.865,Z 927.866,A -85,B 0,C 180,E1 26595.815,E2 26595.815} C_VEL
LIN {X 0,Y 593.194,Z 951.055,A -85,B 0,C 180,E1 26595.251,E2 26595.251} C_VEL
LIN {X 0,Y 591.381,Z 973.312,A -85,B 0,C 180,E1 26594.595,E2 26594.595} C_VEL
LIN {X 0,Y 589.044,Z 998.898,A -85,B 0,C 180,E1 26593.698,E2 26593.698} C_VEL
LIN {X 0,Y 586.233,Z 1026.229,A -85,B 0,C 180,E1 26592.538,E2 26592.538} C_VEL
LIN {X 0,Y 583.88,Z 1047.277,A -85,B 0,C 180,E1 26591.508,E2 26591.508} C_VEL
LIN {X 0,Y 581.555,Z 1066.617,A -85,B 0,C 180,E1 26590.448,E2 26590.448} C_VEL
LIN {X 0,Y 579.076,Z 1086.198,A -85,B 0,C 180,E1 26589.251,E2 26589.251} C_VEL
LIN {X 0,Y 577.031,Z 1101.437,A -85,B 0,C 180,E1 26588.214,E2 26588.214} C_VEL
LIN {X 0,Y 574.569,Z 1116.17,A -85,B 0,C 180,E1 26587.021,E2 26587.021} C_VEL
LIN {X 0,Y 571.344,Z 1134.174,A -85,B 0,C 180,E1 26585.36,E2 26585.36} C_VEL
LIN {X 0,Y 568.414,Z 1150.457,A -85,B 0,C 180,E1 26583.69,E2 26583.69} C_VEL
LIN {X 0,Y 565.503,Z 1167.066,A -85,B 0,C 180,E1 26581.796,E2 26581.796} C_VEL
LIN {X 0,Y 562.145,Z 1186.522,A -85,B 0,C 180,E1 26579.284,E2 26579.284} C_VEL
LIN {X 0,Y 559.856,Z 1200.718,A -85,B 0,C 180,E1 26577.199,E2 26577.199} C_VEL
LIN {X 0,Y 557.925,Z 1213.358,A -85,B 0,C 180,E1 26575.134,E2 26575.134} C_VEL
LIN {X 0,Y 556.076,Z 1227.001,A -85,B 0,C 180,E1 26572.631,E2 26572.631} C_VEL
LIN {X 0,Y 554.55,Z 1239.688,A -85,B 0,C 180,E1 26569.924,E2 26569.924} C_VEL
LIN {X 0,Y 553.553,Z 1249.298,A -85,B 0,C 180,E1 26567.557,E2 26567.557} C_VEL
LIN {X 0,Y 552.914,Z 1257.214,A -85,B 0,C 180,E1 26565.309,E2 26565.309} C_VEL
LIN {X 0,Y 552.368,Z 1265.471,A -85,B 0,C 180,E1 26562.546,E2 26562.546} C_VEL
LIN {X 0,Y 552.057,Z 1271.881,A -85,B 0,C 180,E1 26559.802,E2 26559.802} C_VEL
LIN {X 0,Y 551.96,Z 1276.213,A -85,B 0,C 180,E1 26557.39,E2 26557.39} C_VEL
LIN {X 0,Y 551.922,Z 1279.214,A -85,B 0,C 180,E1 26555.093,E2 26555.093} C_VEL
LIN {X 0,Y 551.909,Z 1281.083,A -85,B 0,C 180,E1 26552.804,E2 26552.804} C_VEL
LIN {X 0,Y 551.878,Z 1281.939,A -85,B 0,C 180,E1 26550.311,E2 26550.311} C_VEL
LIN {X 0,Y 551.907,Z 1281.285,A -85,B 0,C 180,E1 26547.508,E2 26547.508} C_VEL
LIN {X 0,Y 551.922,Z 1279.327,A -85,B 0,C 180,E1 26545.011,E2 26545.011} C_VEL
LIN {X 0,Y 551.965,Z 1276.371,A -85,B 0,C 180,E1 26542.715,E2 26542.715} C_VEL
LIN {X 0,Y 552.034,Z 1272.294,A -85,B 0,C 180,E1 26540.408,E2 26540.408} C_VEL
LIN {X 0,Y 552.3,Z 1266.78,A -85,B 0,C 180,E1 26537.983,E2 26537.983} C_VEL
LIN {X 0,Y 552.837,Z 1258.272,A -85,B 0,C 180,E1 26535.011,E2 26535.011} C_VEL
LIN {X 0,Y 553.475,Z 1250.107,A -85,B 0,C 180,E1 26532.658,E2 26532.658} C_VEL
LIN {X 0,Y 554.389,Z 1241.067,A -85,B 0,C 180,E1 26530.399,E2 26530.399} C_VEL
LIN {X 0,Y 555.578,Z 1230.72,A -85,B 0,C 180,E1 26528.128,E2 26528.128} C_VEL
LIN {X 0,Y 557.477,Z 1216.537,A -85,B 0,C 180,E1 26525.411,E2 26525.411} C_VEL
LIN {X 0,Y 559.646,Z 1202.073,A -85,B 0,C 180,E1 26523.012,E2 26523.012} C_VEL
LIN {X 0,Y 561.77,Z 1188.83,A -85,B 0,C 180,E1 26521.045,E2 26521.045} C_VEL
LIN {X 0,Y 564.545,Z 1172.44,A -85,B 0,C 180,E1 26518.858,E2 26518.858} C_VEL
LIN {X 0,Y 568.029,Z 1152.693,A -85,B 0,C 180,E1 26516.551,E2 26516.551} C_VEL
LIN {X 0,Y 571.014,Z 1136.041,A -85,B 0,C 180,E1 26514.824,E2 26514.824} C_VEL
LIN {X 0,Y 573.923,Z 1119.813,A -85,B 0,C 180,E1 26513.304,E2 26513.304} C_VEL
LIN {X 0,Y 576.378,Z 1105.725,A -85,B 0,C 180,E1 26512.113,E2 26512.113} C_VEL
LIN {X 0,Y 579.188,Z 1087.186,A -85,B 0,C 180,E1 26510.759,E2 26510.759} C_VEL
LIN {X 0,Y 582.004,Z 1068.068,A -85,B 0,C 180,E1 26509.504,E2 26509.504} C_VEL
LIN {X 0,Y 585.014,Z 1046.875,A -85,B 0,C 180,E1 26508.263,E2 26508.263} C_VEL
LIN {X 0,Y 588.655,Z 1019.253,A -85,B 0,C 180,E1 26506.868,E2 26506.868} C_VEL
LIN {X 0,Y 591.21,Z 997.628,A -85,B 0,C 180,E1 26505.937,E2 26505.937} C_VEL
LIN {X 0,Y 593.465,Z 977.202,A -85,B 0,C 180,E1 26505.18,E2 26505.18} C_VEL
LIN {X 0,Y 595.495,Z 956.719,A -85,B 0,C 180,E1 26504.531,E2 26504.531} C_VEL
LIN {X 0,Y 597.262,Z 936.412,A -85,B 0,C 180,E1 26503.994,E2 26503.994} C_VEL
LIN {X 0,Y 598.805,Z 915.64,A -85,B 0,C 180,E1 26503.549,E2 26503.549} C_VEL
LIN {X 0,Y 600.046,Z 892.622,A -85,B 0,C 180,E1 26503.161,E2 26503.161} C_VEL
LIN {X 0,Y 606.432,Z 683.778,A -85,B 0,C 180,E1 26500.172,E2 26500.172} C_VEL
LIN {X 0,Y 613.607,Z 483.242,A -85,B 0,C 180,E1 26497.199,E2 26497.199} C_VEL
LIN {X 0,Y 613.58,Z 479.022,A -85,B 0,C 180,E1 26497.114,E2 26497.114} C_VEL
LIN {X 0,Y 607.504,Z 444.72,A -85,B 0,C 180,E1 26495.695,E2 26495.695} C_VEL
LIN {X 0,Y 595.699,Z 426.505,A -85,B 0,C 180,E1 26493.78,E2 26493.78} C_VEL
LIN {X 0,Y 586.314,Z 412.695,A -85,B 0,C 180,E1 26492.146,E2 26492.146} C_VEL
LIN {X 0,Y 577.787,Z 396.203,A -85,B 0,C 180,E1 26489.438,E2 26489.438} C_VEL
LIN {X 0,Y 569.902,Z 381.763,A -85,B 0,C 180,E1 26486.802,E2 26486.802} C_VEL
LIN {X 0,Y 564.601,Z 372.259,A -85,B 0,C 180,E1 26484.929,E2 26484.929} C_VEL
LIN {X 0,Y 561.604,Z 367.066,A -85,B 0,C 180,E1 26483.838,E2 26483.838} C_VEL
LIN {X 0,Y 558.999,Z 362.347,A -85,B 0,C 180,E1 26482.84,E2 26482.84} C_VEL
LIN {X 0,Y 556.823,Z 358.887,A -85,B 0,C 180,E1 26482.043,E2 26482.043} C_VEL
LIN {X 0,Y 556.152,Z 357.344,A -85,B 0,C 180,E1 26481.738,E2 26481.738} C_VEL
LIN {X 0,Y 553.963,Z 354.13,A -85,B 0,C 180,E1 26480.94,E2 26480.94} C_VEL
LIN {X 0,Y 553.513,Z 352.475,A -85,B 0,C 180,E1 26480.548,E2 26480.548} C_VEL
LIN {X 0,Y 553.497,Z 352.275,A -85,B 0,C 180,E1 26477.234,E2 26477.234} C_VEL
LIN {X 0,Y 553.478,Z 352.284,A -85,B 0,C 180,E1 26473.903,E2 26473.903} C_VEL
LIN {X 0,Y 553.494,Z 352.284,A -85,B 0,C 180,E1 26470.513,E2 26470.513} C_VEL
LIN {X 0,Y 553.509,Z 352.282,A -85,B 0,C 180,E1 26467.16,E2 26467.16} C_VEL
LIN {X 0,Y 553.471,Z 352.287,A -85,B 0,C 180,E1 26463.833,E2 26463.833} C_VEL
LIN {X 0,Y 553.504,Z 352.275,A -85,B 0,C 180,E1 26460.518,E2 26460.518} C_VEL
LIN {X 0,Y 553.478,Z 352.283,A -85,B 0,C 180,E1 26457.204,E2 26457.204} C_VEL
LIN {X 0,Y 553.476,Z 352.285,A -85,B 0,C 180,E1 26453.777,E2 26453.777} C_VEL
LIN {X 0,Y 553.503,Z 352.282,A -85,B 0,C 180,E1 26450.512,E2 26450.512} C_VEL
LIN {X 0,Y 553.464,Z 352.286,A -85,B 0,C 180,E1 26447.161,E2 26447.161} C_VEL
LIN {X 0,Y 553.498,Z 352.282,A -85,B 0,C 180,E1 26443.847,E2 26443.847} C_VEL
LIN {X 0,Y 553.482,Z 352.284,A -85,B 0,C 180,E1 26440.562,E2 26440.562} C_VEL
LIN {X 0,Y 553.463,Z 352.278,A -85,B 0,C 180,E1 26437.144,E2 26437.144} C_VEL
LIN {X 0,Y 553.506,Z 352.276,A -85,B 0,C 180,E1 26433.846,E2 26433.846} C_VEL
LIN {X 0,Y 553.455,Z 352.277,A -85,B 0,C 180,E1 26430.686,E2 26430.686} C_VEL
LIN {X 0,Y 553.499,Z 352.276,A -85,B 0,C 180,E1 26427.429,E2 26427.429} C_VEL
LIN {X 0,Y 553.461,Z 352.277,A -85,B 0,C 180,E1 26424.209,E2 26424.209} C_VEL
LIN {X 0,Y 553.459,Z 352.281,A -85,B 0,C 180,E1 26420.778,E2 26420.778} C_VEL
LIN {X 0,Y 553.491,Z 352.274,A -85,B 0,C 180,E1 26417.634,E2 26417.634} C_VEL
LIN {X 0,Y 553.449,Z 352.283,A -85,B 0,C 180,E1 26414.321,E2 26414.321} C_VEL
LIN {X 0,Y 553.513,Z 352.274,A -85,B 0,C 180,E1 26411.112,E2 26411.112} C_VEL
LIN {X 0,Y 553.445,Z 352.285,A -85,B 0,C 180,E1 26407.898,E2 26407.898} C_VEL
LIN {X 0,Y 553.472,Z 352.285,A -85,B 0,C 180,E1 26404.532,E2 26404.532} C_VEL
LIN {X 0,Y 553.453,Z 352.284,A -85,B 0,C 180,E1 26401.474,E2 26401.474} C_VEL
LIN {X 0,Y 553.45,Z 352.29,A -85,B 0,C 180,E1 26398.134,E2 26398.134} C_VEL
LIN {X 0,Y 553.473,Z 352.284,A -85,B 0,C 180,E1 26395.007,E2 26395.007} C_VEL
LIN {X 0,Y 553.437,Z 352.288,A -85,B 0,C 180,E1 26391.738,E2 26391.738} C_VEL
LIN {X 0,Y 553.497,Z 352.28,A -85,B 0,C 180,E1 26388.538,E2 26388.538} C_VEL
LIN {X 0,Y 553.43,Z 352.282,A -85,B 0,C 180,E1 26385.294,E2 26385.294} C_VEL
LIN {X 0,Y 553.486,Z 352.279,A -85,B 0,C 180,E1 26382.096,E2 26382.096} C_VEL
LIN {X 0,Y 553.429,Z 352.293,A -85,B 0,C 180,E1 26378.939,E2 26378.939} C_VEL
LIN {X 0,Y 553.452,Z 352.283,A -85,B 0,C 180,E1 26377.692,E2 26377.692} C_VEL
LIN {X 0,Y 552.416,Z 352.413,A -85,B 0,C 180,E1 26376.895,E2 26376.895} C_VEL
LIN {X 0,Y 546.061,Z 353.204,A -85,B 0,C 180,E1 26374.655,E2 26374.655} C_VEL
LIN {X 0,Y 545.547,Z 353.273,A -85,B 0,C 180,E1 26374.073,E2 26374.073} C_VEL
LIN {X 0,Y 545.482,Z 353.278,A -85,B 0,C 180,E1 26370.84,E2 26370.84} C_VEL
LIN {X 0,Y 545.569,Z 353.525,A -85,B 0,C 180,E1 26368.057,E2 26368.057} C_VEL
LIN {X 0,Y 545.886,Z 354.761,A -85,B 0,C 180,E1 26367.796,E2 26367.796} C_VEL
LIN {X 0,Y 547.77,Z 357.899,A -85,B 0,C 180,E1 26367.332,E2 26367.332} C_VEL
LIN {X 0,Y 550.403,Z 360.028,A -85,B 0,C 180,E1 26366.798,E2 26366.798} C_VEL
LIN {X 0,Y 552.824,Z 363.787,A -85,B 0,C 180,E1 26366.267,E2 26366.267} C_VEL
LIN {X 0,Y 555.354,Z 366.233,A -85,B 0,C 180,E1 26365.767,E2 26365.767} C_VEL
LIN {X 0,Y 558.281,Z 370.282,A -85,B 0,C 180,E1 26365.171,E2 26365.171} C_VEL
LIN {X 0,Y 560.641,Z 372.563,A -85,B 0,C 180,E1 26364.73,E2 26364.73} C_VEL
LIN {X 0,Y 564.143,Z 376.945,A -85,B 0,C 180,E1 26364.049,E2 26364.049} C_VEL
LIN {X 0,Y 570.526,Z 385.022,A -85,B 0,C 180,E1 26362.852,E2 26362.852} C_VEL
LIN {X 0,Y 579.732,Z 396.558,A -85,B 0,C 180,E1 26361.221,E2 26361.221} C_VEL
LIN {X 0,Y 591.15,Z 411.373,A -85,B 0,C 180,E1 26359.335,E2 26359.335} C_VEL
LIN {X 0,Y 602.118,Z 426.313,A -85,B 0,C 180,E1 26357.63,E2 26357.63} C_VEL
LIN {X 0,Y 606.446,Z 432.702,A -85,B 0,C 180,E1 26356.98,E2 26356.98} C_VEL
LIN {X 0,Y 598.725,Z 640.215,A -85,B 0,C 180,E1 26353.913,E2 26353.913} C_VEL
LIN {X 0,Y 594.59,Z 761.481,A -85,B 0,C 180,E1 26352.151,E2 26352.151} C_VEL
LIN {X 0,Y 592.858,Z 789.313,A -85,B 0,C 180,E1 26351.603,E2 26351.603} C_VEL
LIN {X 0,Y 590.719,Z 814.052,A -85,B 0,C 180,E1 26350.943,E2 26350.943} C_VEL
LIN {X 0,Y 588.551,Z 835.142,A -85,B 0,C 180,E1 26350.253,E2 26350.253} C_VEL
LIN {X 0,Y 585.942,Z 857.228,A -85,B 0,C 180,E1 26349.393,E2 26349.393} C_VEL
LIN {X 0,Y 582.397,Z 883.191,A -85,B 0,C 180,E1 26348.185,E2 26348.185} C_VEL
LIN {X 0,Y 578.848,Z 906.127,A -85,B 0,C 180,E1 26346.914,E2 26346.914} C_VEL
LIN {X 0,Y 574.981,Z 929.095,A -85,B 0,C 180,E1 26345.436,E2 26345.436} C_VEL
LIN {X 0,Y 570.865,Z 951.71,A -85,B 0,C 180,E1 26343.739,E2 26343.739} C_VEL
LIN {X 0,Y 567.084,Z 971.553,A -85,B 0,C 180,E1 26342.03,E2 26342.03} C_VEL
LIN {X 0,Y 562.216,Z 996.65,A -85,B 0,C 180,E1 26339.545,E2 26339.545} C_VEL
LIN {X 0,Y 558.658,Z 1015.468,A -85,B 0,C 180,E1 26337.403,E2 26337.403} C_VEL
LIN {X 0,Y 555.29,Z 1033.986,A -85,B 0,C 180,E1 26335.015,E2 26335.015} C_VEL
LIN {X 0,Y 552.394,Z 1050.867,A -85,B 0,C 180,E1 26332.542,E2 26332.542} C_VEL
LIN {X 0,Y 549.871,Z 1066.699,A -85,B 0,C 180,E1 26329.883,E2 26329.883} C_VEL
LIN {X 0,Y 547.895,Z 1080.544,A -85,B 0,C 180,E1 26327.192,E2 26327.192} C_VEL
LIN {X 0,Y 546.353,Z 1093.154,A -85,B 0,C 180,E1 26324.356,E2 26324.356} C_VEL
LIN {X 0,Y 545.293,Z 1103.674,A -85,B 0,C 180,E1 26321.572,E2 26321.572} C_VEL
LIN {X 0,Y 544.631,Z 1112.161,A -85,B 0,C 180,E1 26318.885,E2 26318.885} C_VEL
LIN {X 0,Y 544.191,Z 1119.203,A -85,B 0,C 180,E1 26316.143,E2 26316.143} C_VEL
LIN {X 0,Y 544.012,Z 1124.412,A -85,B 0,C 180,E1 26313.589,E2 26313.589} C_VEL
LIN {X 0,Y 543.937,Z 1128.258,A -85,B 0,C 180,E1 26310.978,E2 26310.978} C_VEL
LIN {X 0,Y 543.919,Z 1130.823,A -85,B 0,C 180,E1 26308.313,E2 26308.313} C_VEL
LIN {X 0,Y 543.906,Z 1131.873,A -85,B 0,C 180,E1 26305.712,E2 26305.712} C_VEL
LIN {X 0,Y 543.87,Z 1131.617,A -85,B 0,C 180,E1 26303.054,E2 26303.054} C_VEL
LIN {X 0,Y 543.919,Z 1129.895,A -85,B 0,C 180,E1 26300.443,E2 26300.443} C_VEL
LIN {X 0,Y 543.974,Z 1126.542,A -85,B 0,C 180,E1 26297.655,E2 26297.655} C_VEL
LIN {X 0,Y 544.128,Z 1121.624,A -85,B 0,C 180,E1 26294.859,E2 26294.859} C_VEL
LIN {X 0,Y 544.438,Z 1114.802,A -85,B 0,C 180,E1 26291.978,E2 26291.978} C_VEL
LIN {X 0,Y 544.986,Z 1106.836,A -85,B 0,C 180,E1 26289.291,E2 26289.291} C_VEL
LIN {X 0,Y 545.856,Z 1097.854,A -85,B 0,C 180,E1 26286.733,E2 26286.733} C_VEL
LIN {X 0,Y 547.13,Z 1086.431,A -85,B 0,C 180,E1 26283.982,E2 26283.982} C_VEL
LIN {X 0,Y 548.89,Z 1073.219,A -85,B 0,C 180,E1 26281.253,E2 26281.253} C_VEL
LIN {X 0,Y 551.087,Z 1058.748,A -85,B 0,C 180,E1 26278.648,E2 26278.648} C_VEL
LIN {X 0,Y 553.862,Z 1042.306,A -85,B 0,C 180,E1 26276.066,E2 26276.066} C_VEL
LIN {X 0,Y 557.037,Z 1024.361,A -85,B 0,C 180,E1 26273.61,E2 26273.61} C_VEL
LIN {X 0,Y 560.471,Z 1005.825,A -85,B 0,C 180,E1 26271.381,E2 26271.381} C_VEL
LIN {X 0,Y 564.601,Z 984.048,A -85,B 0,C 180,E1 26269.077,E2 26269.077} C_VEL
LIN {X 0,Y 568.742,Z 963.806,A -85,B 0,C 180,E1 26267.15,E2 26267.15} C_VEL
LIN {X 0,Y 572.62,Z 943.521,A -85,B 0,C 180,E1 26265.488,E2 26265.488} C_VEL
LIN {X 0,Y 575.852,Z 925.244,A -85,B 0,C 180,E1 26264.18,E2 26264.18} C_VEL
LIN {X 0,Y 579.101,Z 905.338,A -85,B 0,C 180,E1 26262.931,E2 26262.931} C_VEL
LIN {X 0,Y 582.55,Z 881.312,A -85,B 0,C 180,E1 26261.647,E2 26261.647} C_VEL
LIN {X 0,Y 585.019,Z 861.306,A -85,B 0,C 180,E1 26260.739,E2 26260.739} C_VEL
LIN {X 0,Y 587.108,Z 841.828,A -85,B 0,C 180,E1 26259.982,E2 26259.982} C_VEL
LIN {X 0,Y 588.96,Z 821.338,A -85,B 0,C 180,E1 26259.307,E2 26259.307} C_VEL
LIN {X 0,Y 590.837,Z 795.883,A -85,B 0,C 180,E1 26258.627,E2 26258.627} C_VEL
LIN {X 0,Y 592.066,Z 769.874,A -85,B 0,C 180,E1 26258.121,E2 26258.121} C_VEL
LIN {X 0,Y 597.24,Z 612.953,A -85,B 0,C 180,E1 26255.827,E2 26255.827} C_VEL
LIN {X 0,Y 601.834,Z 515.911,A -85,B 0,C 180,E1 26254.292,E2 26254.292} C_VEL
LIN {X 0,Y 607.052,Z 436.549,A -85,B 0,C 180,E1 26252.944,E2 26252.944} C_VEL
LIN {X 0,Y 607.249,Z 432.227,A -85,B 0,C 180,E1 26252.847,E2 26252.847} C_VEL
LIN {X 0,Y 602.808,Z 423.089,A -85,B 0,C 180,E1 26251.707,E2 26251.707} C_VEL
LIN {X 0,Y 600.164,Z 417.343,A -85,B 0,C 180,E1 26250.781,E2 26250.781} C_VEL
LIN {X 0,Y 598.812,Z 414.126,A -85,B 0,C 180,E1 26250.103,E2 26250.103} C_VEL
LIN {X 0,Y 598.036,Z 412.115,A -85,B 0,C 180,E1 26249.562,E2 26249.562} C_VEL
LIN {X 0,Y 597.585,Z 411.459,A -85,B 0,C 180,E1 26249.132,E2 26249.132} C_VEL
LIN {X 0,Y 596.677,Z 414.326,A -85,B 0,C 180,E1 26248.392,E2 26248.392} C_VEL
LIN {X 0,Y 596.431,Z 420.176,A -85,B 0,C 180,E1 26247.386,E2 26247.386} C_VEL
LIN {X 0,Y 597.08,Z 427.059,A -85,B 0,C 180,E1 26246.497,E2 26246.497} C_VEL
LIN {X 0,Y 599.589,Z 439.312,A -85,B 0,C 180,E1 26245.212,E2 26245.212} C_VEL
LIN {X 0,Y 601.377,Z 444.892,A -85,B 0,C 180,E1 26244.647,E2 26244.647} C_VEL
LIN {X 0,Y 603.239,Z 471.258,A -85,B 0,C 180,E1 26243.523,E2 26243.523} C_VEL
LIN {X 0,Y 604.514,Z 482.029,A -85,B 0,C 180,E1 26243.063,E2 26243.063} C_VEL
LIN {X 0,Y 599.926,Z 567.719,A -85,B 0,C 180,E1 26241.634,E2 26241.634} C_VEL
LIN {X 0,Y 596.044,Z 667.207,A -85,B 0,C 180,E1 26240.087,E2 26240.087} C_VEL
LIN {X 0,Y 592.769,Z 786.241,A -85,B 0,C 180,E1 26238.38,E2 26238.38} C_VEL
LIN {X 0,Y 590.292,Z 893.361,A -85,B 0,C 180,E1 26236.904,E2 26236.904} C_VEL
LIN {X 0,Y 588.493,Z 923.972,A -85,B 0,C 180,E1 26236.338,E2 26236.338} C_VEL
LIN {X 0,Y 586.685,Z 948.018,A -85,B 0,C 180,E1 26235.757,E2 26235.757} C_VEL
LIN {X 0,Y 584.791,Z 970.255,A -85,B 0,C 180,E1 26235.104,E2 26235.104} C_VEL
LIN {X 0,Y 582.428,Z 995.52,A -85,B 0,C 180,E1 26234.221,E2 26234.221} C_VEL
LIN {X 0,Y 579.487,Z 1023.418,A -85,B 0,C 180,E1 26233.046,E2 26233.046} C_VEL
LIN {X 0,Y 576.966,Z 1045.009,A -85,B 0,C 180,E1 26231.985,E2 26231.985} C_VEL
LIN {X 0,Y 574.667,Z 1063.589,A -85,B 0,C 180,E1 26230.962,E2 26230.962} C_VEL
LIN {X 0,Y 572.278,Z 1081.914,A -85,B 0,C 180,E1 26229.845,E2 26229.845} C_VEL
LIN {X 0,Y 569.703,Z 1100.606,A -85,B 0,C 180,E1 26228.582,E2 26228.582} C_VEL
LIN {X 0,Y 567.084,Z 1118.897,A -85,B 0,C 180,E1 26227.212,E2 26227.212} C_VEL
LIN {X 0,Y 565.114,Z 1131.031,A -85,B 0,C 180,E1 26226.162,E2 26226.162} C_VEL
LIN {X 0,Y 561.763,Z 1148.771,A -85,B 0,C 180,E1 26224.348,E2 26224.348} C_VEL
LIN {X 0,Y 558.844,Z 1164.388,A -85,B 0,C 180,E1 26222.571,E2 26222.571} C_VEL
LIN {X 0,Y 555.992,Z 1180.046,A -85,B 0,C 180,E1 26220.593,E2 26220.593} C_VEL
LIN {X 0,Y 552.739,Z 1198.57,A -85,B 0,C 180,E1 26217.938,E2 26217.938} C_VEL
LIN {X 0,Y 550.565,Z 1212.086,A -85,B 0,C 180,E1 26215.724,E2 26215.724} C_VEL
LIN {X 0,Y 548.77,Z 1224.134,A -85,B 0,C 180,E1 26213.517,E2 26213.517} C_VEL
LIN {X 0,Y 547.043,Z 1237.371,A -85,B 0,C 180,E1 26210.768,E2 26210.768} C_VEL
LIN {X 0,Y 545.78,Z 1248.487,A -85,B 0,C 180,E1 26208.036,E2 26208.036} C_VEL
LIN {X 0,Y 545.033,Z 1256.507,A -85,B 0,C 180,E1 26205.754,E2 26205.754} C_VEL
LIN {X 0,Y 544.534,Z 1263.351,A -85,B 0,C 180,E1 26203.485,E2 26203.485} C_VEL
LIN {X 0,Y 544.191,Z 1269.579,A -85,B 0,C 180,E1 26201.016,E2 26201.016} C_VEL
LIN {X 0,Y 543.985,Z 1275.251,A -85,B 0,C 180,E1 26198.136,E2 26198.136} C_VEL
LIN {X 0,Y 543.931,Z 1278.757,A -85,B 0,C 180,E1 26195.591,E2 26195.591} C_VEL
LIN {X 0,Y 543.911,Z 1280.811,A -85,B 0,C 180,E1 26193.267,E2 26193.267} C_VEL
LIN {X 0,Y 543.886,Z 1281.758,A -85,B 0,C 180,E1 26191.159,E2 26191.159} C_VEL
LIN {X 0,Y 543.872,Z 1281.804,A -85,B 0,C 180,E1 26189.052,E2 26189.052} C_VEL
LIN {X 0,Y 543.91,Z 1280.946,A -85,B 0,C 180,E1 26186.944,E2 26186.944} C_VEL
LIN {X 0,Y 543.925,Z 1279.097,A -85,B 0,C 180,E1 26184.726,E2 26184.726} C_VEL
LIN {X 0,Y 543.959,Z 1276.049,A -85,B 0,C 180,E1 26182.395,E2 26182.395} C_VEL
LIN {X 0,Y 544.115,Z 1271.465,A -85,B 0,C 180,E1 26179.839,E2 26179.839} C_VEL
LIN {X 0,Y 544.492,Z 1264.259,A -85,B 0,C 180,E1 26176.838,E2 26176.838} C_VEL
LIN {X 0,Y 545.009,Z 1256.858,A -85,B 0,C 180,E1 26174.354,E2 26174.354} C_VEL
LIN {X 0,Y 545.736,Z 1248.891,A -85,B 0,C 180,E1 26172.073,E2 26172.073} C_VEL
LIN {X 0,Y 546.871,Z 1238.771,A -85,B 0,C 180,E1 26169.561,E2 26169.561} C_VEL
LIN {X 0,Y 548.616,Z 1225.286,A -85,B 0,C 180,E1 26166.703,E2 26166.703} C_VEL
LIN {X 0,Y 550.462,Z 1212.723,A -85,B 0,C 180,E1 26164.386,E2 26164.386} C_VEL
LIN {X 0,Y 552.548,Z 1199.688,A -85,B 0,C 180,E1 26162.239,E2 26162.239} C_VEL
LIN {X 0,Y 555.574,Z 1182.583,A -85,B 0,C 180,E1 26159.74,E2 26159.74} C_VEL
LIN {X 0,Y 558.699,Z 1165.213,A -85,B 0,C 180,E1 26157.527,E2 26157.527} C_VEL
LIN {X 0,Y 561.574,Z 1149.785,A -85,B 0,C 180,E1 26155.762,E2 26155.762} C_VEL
LIN {X 0,Y 564.69,Z 1133.263,A -85,B 0,C 180,E1 26154.057,E2 26154.057} C_VEL
LIN {X 0,Y 566.704,Z 1121.708,A -85,B 0,C 180,E1 26153.012,E2 26153.012} C_VEL
LIN {X 0,Y 569.686,Z 1103.284,A -85,B 0,C 180,E1 26151.518,E2 26151.518} C_VEL
LIN {X 0,Y 572.673,Z 1084.559,A -85,B 0,C 180,E1 26150.15,E2 26150.15} C_VEL
LIN {X 0,Y 575.763,Z 1064.553,A -85,B 0,C 180,E1 26148.839,E2 26148.839} C_VEL
LIN {X 0,Y 579.494,Z 1039.08,A -85,B 0,C 180,E1 26147.372,E2 26147.372} C_VEL
LIN {X 0,Y 582.598,Z 1016.026,A -85,B 0,C 180,E1 26146.24,E2 26146.24} C_VEL
LIN {X 0,Y 585.085,Z 996.059,A -85,B 0,C 180,E1 26145.382,E2 26145.382} C_VEL
LIN {X 0,Y 587.381,Z 976.112,A -85,B 0,C 180,E1 26144.639,E2 26144.639} C_VEL
LIN {X 0,Y 589.505,Z 955.77,A -85,B 0,C 180,E1 26143.993,E2 26143.993} C_VEL
LIN {X 0,Y 591.39,Z 935.046,A -85,B 0,C 180,E1 26143.443,E2 26143.443} C_VEL
LIN {X 0,Y 593.056,Z 913.492,A -85,B 0,C 180,E1 26142.983,E2 26142.983} C_VEL
LIN {X 0,Y 594.528,Z 885.67,A -85,B 0,C 180,E1 26142.523,E2 26142.523} C_VEL
LIN {X 0,Y 600.894,Z 687.577,A -85,B 0,C 180,E1 26139.664,E2 26139.664} C_VEL
LIN {X 0,Y 608.247,Z 491.167,A -85,B 0,C 180,E1 26136.733,E2 26136.733} C_VEL
LIN {X 0,Y 608.476,Z 481.152,A -85,B 0,C 180,E1 26136.562,E2 26136.562} C_VEL
LIN {X 0,Y 603.071,Z 449.603,A -85,B 0,C 180,E1 26135.239,E2 26135.239} C_VEL
LIN {X 0,Y 589.63,Z 428.968,A -85,B 0,C 180,E1 26133.009,E2 26133.009} C_VEL
LIN {X 0,Y 577.112,Z 410.753,A -85,B 0,C 180,E1 26130.738,E2 26130.738} C_VEL
LIN {X 0,Y 569.121,Z 395.73,A -85,B 0,C 180,E1 26128.121,E2 26128.121} C_VEL
LIN {X 0,Y 562.572,Z 383.496,A -85,B 0,C 180,E1 26125.814,E2 26125.814} C_VEL
LIN {X 0,Y 556.497,Z 372.959,A -85,B 0,C 180,E1 26123.621,E2 26123.621} C_VEL
LIN {X 0,Y 553.887,Z 368.289,A -85,B 0,C 180,E1 26122.614,E2 26122.614} C_VEL
LIN {X 0,Y 551.799,Z 364.677,A -85,B 0,C 180,E1 26121.806,E2 26121.806} C_VEL
LIN {X 0,Y 550.448,Z 362.601,A -85,B 0,C 180,E1 26121.303,E2 26121.303} C_VEL
LIN {X 0,Y 548.027,Z 358.164,A -85,B 0,C 180,E1 26120.283,E2 26120.283} C_VEL
LIN {X 0,Y 545.977,Z 355.001,A -85,B 0,C 180,E1 26119.47,E2 26119.47} C_VEL
LIN {X 0,Y 545.586,Z 353.452,A -85,B 0,C 180,E1 26119.095,E2 26119.095} C_VEL
LIN {X 0,Y 545.55,Z 353.261,A -85,B 0,C 180,E1 26115.739,E2 26115.739} C_VEL
LIN {X 0,Y 545.541,Z 353.258,A -85,B 0,C 180,E1 26112.275,E2 26112.275} C_VEL
LIN {X 0,Y 545.56,Z 353.256,A -85,B 0,C 180,E1 26108.94,E2 26108.94} C_VEL
LIN {X 0,Y 545.534,Z 353.259,A -85,B 0,C 180,E1 26105.68,E2 26105.68} C_VEL
LIN {X 0,Y 545.555,Z 353.258,A -85,B 0,C 180,E1 26102.311,E2 26102.311} C_VEL
LIN {X 0,Y 545.564,Z 353.27,A -85,B 0,C 180,E1 26098.95,E2 26098.95} C_VEL
LIN {X 0,Y 545.529,Z 353.273,A -85,B 0,C 180,E1 26095.585,E2 26095.585} C_VEL
LIN {X 0,Y 545.566,Z 353.275,A -85,B 0,C 180,E1 26092.205,E2 26092.205} C_VEL
LIN {X 0,Y 545.539,Z 353.272,A -85,B 0,C 180,E1 26088.904,E2 26088.904} C_VEL
LIN {X 0,Y 545.528,Z 353.274,A -85,B 0,C 180,E1 26085.457,E2 26085.457} C_VEL
LIN {X 0,Y 545.566,Z 353.262,A -85,B 0,C 180,E1 26082.177,E2 26082.177} C_VEL
LIN {X 0,Y 545.524,Z 353.275,A -85,B 0,C 180,E1 26078.833,E2 26078.833} C_VEL
LIN {X 0,Y 545.543,Z 353.276,A -85,B 0,C 180,E1 26075.414,E2 26075.414} C_VEL
LIN {X 0,Y 545.564,Z 353.272,A -85,B 0,C 180,E1 26072.053,E2 26072.053} C_VEL
LIN {X 0,Y 545.518,Z 353.278,A -85,B 0,C 180,E1 26068.754,E2 26068.754} C_VEL
LIN {X 0,Y 545.566,Z 353.276,A -85,B 0,C 180,E1 26065.506,E2 26065.506} C_VEL
LIN {X 0,Y 545.521,Z 353.276,A -85,B 0,C 180,E1 26062.183,E2 26062.183} C_VEL
LIN {X 0,Y 545.521,Z 353.271,A -85,B 0,C 180,E1 26058.711,E2 26058.711} C_VEL
LIN {X 0,Y 545.561,Z 353.268,A -85,B 0,C 180,E1 26055.416,E2 26055.416} C_VEL
LIN {X 0,Y 545.507,Z 353.271,A -85,B 0,C 180,E1 26052.133,E2 26052.133} C_VEL
LIN {X 0,Y 545.551,Z 353.265,A -85,B 0,C 180,E1 26048.815,E2 26048.815} C_VEL
LIN {X 0,Y 545.512,Z 353.268,A -85,B 0,C 180,E1 26045.652,E2 26045.652} C_VEL
LIN {X 0,Y 545.512,Z 353.269,A -85,B 0,C 180,E1 26042.234,E2 26042.234} C_VEL
LIN {X 0,Y 545.532,Z 353.263,A -85,B 0,C 180,E1 26039.179,E2 26039.179} C_VEL
LIN {X 0,Y 545.501,Z 353.271,A -85,B 0,C 180,E1 26035.842,E2 26035.842} C_VEL
LIN {X 0,Y 545.568,Z 353.265,A -85,B 0,C 180,E1 26032.522,E2 26032.522} C_VEL
LIN {X 0,Y 545.499,Z 353.28,A -85,B 0,C 180,E1 26029.265,E2 26029.265} C_VEL
LIN {X 0,Y 545.509,Z 353.274,A -85,B 0,C 180,E1 26025.849,E2 26025.849} C_VEL
LIN {X 0,Y 545.502,Z 353.274,A -85,B 0,C 180,E1 26022.922,E2 26022.922} C_VEL
LIN {X 0,Y 545.495,Z 353.274,A -85,B 0,C 180,E1 26019.495,E2 26019.495} C_VEL
LIN {X 0,Y 545.513,Z 353.277,A -85,B 0,C 180,E1 26016.525,E2 26016.525} C_VEL
LIN {X 0,Y 545.547,Z 353.273,A -85,B 0,C 180,E1 26014.073,E2 26014.073} C_VEL
LIN {X 0,Y 544.55,Z 353.406,A -85,B 0,C 180,E1 26013.264,E2 26013.264} C_VEL
LIN {X 0,Y 538.063,Z 354.205,A -85,B 0,C 180,E1 26010.993,E2 26010.993} C_VEL
LIN {X 0,Y 537.564,Z 354.261,A -85,B 0,C 180,E1 26010.4,E2 26010.4} C_VEL
LIN {X 0,Y 537.599,Z 354.386,A -85,B 0,C 180,E1 26009.574,E2 26009.574} C_VEL
LIN {X 0,Y 537.883,Z 355.742,A -85,B 0,C 180,E1 26009.281,E2 26009.281} C_VEL
LIN {X 0,Y 539.561,Z 358.657,A -85,B 0,C 180,E1 26008.859,E2 26008.859} C_VEL
LIN {X 0,Y 542.683,Z 361.143,A -85,B 0,C 180,E1 26008.179,E2 26008.179} C_VEL
LIN {X 0,Y 544.99,Z 364.843,A -85,B 0,C 180,E1 26007.634,E2 26007.634} C_VEL
LIN {X 0,Y 547.681,Z 367.324,A -85,B 0,C 180,E1 26007.07,E2 26007.07} C_VEL
LIN {X 0,Y 550.609,Z 371.368,A -85,B 0,C 180,E1 26006.434,E2 26006.434} C_VEL
LIN {X 0,Y 552.478,Z 373.292,A -85,B 0,C 180,E1 26006.057,E2 26006.057} C_VEL
LIN {X 0,Y 555.909,Z 377.732,A -85,B 0,C 180,E1 26005.358,E2 26005.358} C_VEL
LIN {X 0,Y 557.968,Z 379.937,A -85,B 0,C 180,E1 26004.963,E2 26004.963} C_VEL
LIN {X 0,Y 563.105,Z 386.412,A -85,B 0,C 180,E1 26003.964,E2 26003.964} C_VEL
LIN {X 0,Y 567.603,Z 392.015,A -85,B 0,C 180,E1 26003.12,E2 26003.12} C_VEL
LIN {X 0,Y 579.197,Z 406.564,A -85,B 0,C 180,E1 26001.062,E2 26001.062} C_VEL
LIN {X 0,Y 594.125,Z 426.459,A -85,B 0,C 180,E1 25998.632,E2 25998.632} C_VEL
LIN {X 0,Y 601.305,Z 436.852,A -85,B 0,C 180,E1 25997.517,E2 25997.517} C_VEL
LIN {X 0,Y 593.389,Z 638.545,A -85,B 0,C 180,E1 25994.51,E2 25994.51} C_VEL
LIN {X 0,Y 588.927,Z 762.518,A -85,B 0,C 180,E1 25992.689,E2 25992.689} C_VEL
LIN {X 0,Y 587.104,Z 790.635,A -85,B 0,C 180,E1 25992.129,E2 25992.129} C_VEL
LIN {X 0,Y 584.909,Z 815.186,A -85,B 0,C 180,E1 25991.468,E2 25991.468} C_VEL
LIN {X 0,Y 582.727,Z 835.736,A -85,B 0,C 180,E1 25990.791,E2 25990.791} C_VEL
LIN {X 0,Y 580.245,Z 856.114,A -85,B 0,C 180,E1 25989.998,E2 25989.998} C_VEL
LIN {X 0,Y 577.269,Z 877.937,A -85,B 0,C 180,E1 25989.005,E2 25989.005} C_VEL
LIN {X 0,Y 573.186,Z 903.95,A -85,B 0,C 180,E1 25987.602,E2 25987.602} C_VEL
LIN {X 0,Y 569.456,Z 925.526,A -85,B 0,C 180,E1 25986.236,E2 25986.236} C_VEL
LIN {X 0,Y 565.406,Z 947.359,A -85,B 0,C 180,E1 25984.646,E2 25984.646} C_VEL
LIN {X 0,Y 561.218,Z 968.46,A -85,B 0,C 180,E1 25982.865,E2 25982.865} C_VEL
LIN {X 0,Y 557.143,Z 988.458,A -85,B 0,C 180,E1 25980.928,E2 25980.928} C_VEL
LIN {X 0,Y 552.825,Z 1009.341,A -85,B 0,C 180,E1 25978.608,E2 25978.608} C_VEL
LIN {X 0,Y 549.209,Z 1027.773,A -85,B 0,C 180,E1 25976.307,E2 25976.307} C_VEL
LIN {X 0,Y 546.015,Z 1044.958,A -85,B 0,C 180,E1 25973.861,E2 25973.861} C_VEL
LIN {X 0,Y 543.192,Z 1061.046,A -85,B 0,C 180,E1 25971.255,E2 25971.255} C_VEL
LIN {X 0,Y 540.912,Z 1075.552,A -85,B 0,C 180,E1 25968.566,E2 25968.566} C_VEL
LIN {X 0,Y 539.103,Z 1088.44,A -85,B 0,C 180,E1 25965.784,E2 25965.784} C_VEL
LIN {X 0,Y 537.823,Z 1099.4,A -85,B 0,C 180,E1 25963.024,E2 25963.024} C_VEL
LIN {X 0,Y 536.93,Z 1108.856,A -85,B 0,C 180,E1 25960.226,E2 25960.226} C_VEL
LIN {X 0,Y 536.373,Z 1116.245,A -85,B 0,C 180,E1 25957.56,E2 25957.56} C_VEL
LIN {X 0,Y 536.094,Z 1122.649,A -85,B 0,C 180,E1 25954.663,E2 25954.663} C_VEL
LIN {X 0,Y 535.958,Z 1127.279,A -85,B 0,C 180,E1 25951.869,E2 25951.869} C_VEL
LIN {X 0,Y 535.922,Z 1130.219,A -85,B 0,C 180,E1 25949.141,E2 25949.141} C_VEL
LIN {X 0,Y 535.898,Z 1131.747,A -85,B 0,C 180,E1 25946.417,E2 25946.417} C_VEL
LIN {X 0,Y 535.902,Z 1131.824,A -85,B 0,C 180,E1 25943.884,E2 25943.884} C_VEL
LIN {X 0,Y 535.916,Z 1130.504,A -85,B 0,C 180,E1 25941.106,E2 25941.106} C_VEL
LIN {X 0,Y 535.948,Z 1127.851,A -85,B 0,C 180,E1 25938.491,E2 25938.491} C_VEL
LIN {X 0,Y 536.057,Z 1123.479,A -85,B 0,C 180,E1 25935.692,E2 25935.692} C_VEL
LIN {X 0,Y 536.335,Z 1117.68,A -85,B 0,C 180,E1 25932.928,E2 25932.928} C_VEL
LIN {X 0,Y 536.828,Z 1110.35,A -85,B 0,C 180,E1 25930.192,E2 25930.192} C_VEL
LIN {X 0,Y 537.629,Z 1101.171,A -85,B 0,C 180,E1 25927.373,E2 25927.373} C_VEL
LIN {X 0,Y 538.809,Z 1090.822,A -85,B 0,C 180,E1 25924.684,E2 25924.684} C_VEL
LIN {X 0,Y 540.431,Z 1078.797,A -85,B 0,C 180,E1 25922.015,E2 25922.015} C_VEL
LIN {X 0,Y 542.552,Z 1065.055,A -85,B 0,C 180,E1 25919.366,E2 25919.366} C_VEL
LIN {X 0,Y 545.204,Z 1049.462,A -85,B 0,C 180,E1 25916.741,E2 25916.741} C_VEL
LIN {X 0,Y 548.349,Z 1032.543,A -85,B 0,C 180,E1 25914.244,E2 25914.244} C_VEL
LIN {X 0,Y 551.848,Z 1014.151,A -85,B 0,C 180,E1 25911.875,E2 25911.875} C_VEL
LIN {X 0,Y 556.94,Z 990.272,A -85,B 0,C 180,E1 25909.134,E2 25909.134} C_VEL
LIN {X 0,Y 560.677,Z 972.691,A -85,B 0,C 180,E1 25907.381,E2 25907.381} C_VEL
LIN {X 0,Y 564.593,Z 953.508,A -85,B 0,C 180,E1 25905.697,E2 25905.697} C_VEL
LIN {X 0,Y 568.704,Z 931.344,A -85,B 0,C 180,E1 25904.029,E2 25904.029} C_VEL
LIN {X 0,Y 571.883,Z 912.695,A -85,B 0,C 180,E1 25902.813,E2 25902.813} C_VEL
LIN {X 0,Y 574.773,Z 894.115,A -85,B 0,C 180,E1 25901.752,E2 25901.752} C_VEL
LIN {X 0,Y 577.584,Z 873.882,A -85,B 0,C 180,E1 25900.744,E2 25900.744} C_VEL
LIN {X 0,Y 580.489,Z 848.784,A -85,B 0,C 180,E1 25899.691,E2 25899.691} C_VEL
LIN {X 0,Y 582.577,Z 826.727,A -85,B 0,C 180,E1 25898.933,E2 25898.933} C_VEL
LIN {X 0,Y 584.209,Z 805.93,A -85,B 0,C 180,E1 25898.345,E2 25898.345} C_VEL
LIN {X 0,Y 585.635,Z 782.087,A -85,B 0,C 180,E1 25897.809,E2 25897.809} C_VEL
LIN {X 0,Y 586.982,Z 745.469,A -85,B 0,C 180,E1 25897.232,E2 25897.232} C_VEL
LIN {X 0,Y 591.284,Z 625.63,A -85,B 0,C 180,E1 25895.451,E2 25895.451} C_VEL
LIN {X 0,Y 596.29,Z 529.349,A -85,B 0,C 180,E1 25893.895,E2 25893.895} C_VEL
LIN {X 0,Y 601.757,Z 453.061,A -85,B 0,C 180,E1 25892.572,E2 25892.572} C_VEL
LIN {X 0,Y 603.122,Z 436.563,A -85,B 0,C 180,E1 25892.263,E2 25892.263} C_VEL
LIN {X 0,Y 599.589,Z 428.337,A -85,B 0,C 180,E1 25891.174,E2 25891.174} C_VEL
LIN {X 0,Y 597.302,Z 422.496,A -85,B 0,C 180,E1 25890.126,E2 25890.126} C_VEL
LIN {X 0,Y 596.337,Z 419.68,A -85,B 0,C 180,E1 25889.354,E2 25889.354} C_VEL
LIN {X 0,Y 596.131,Z 419.55,A -85,B 0,C 180,E1 25889.178,E2 25889.178} C_VEL
LIN {X 0,Y 594.942,Z 423.702,A -85,B 0,C 180,E1 25888.29,E2 25888.29} C_VEL
LIN {X 0,Y 594.678,Z 430.374,A -85,B 0,C 180,E1 25887.277,E2 25887.277} C_VEL
LIN {X 0,Y 595.817,Z 441.664,A -85,B 0,C 180,E1 25886.025,E2 25886.025} C_VEL
LIN {X 0,Y 597.754,Z 449.79,A -85,B 0,C 180,E1 25885.177,E2 25885.177} C_VEL
LIN {X 0,Y 598.929,Z 474.319,A -85,B 0,C 180,E1 25884.096,E2 25884.096} C_VEL
LIN {X 0,Y 599.853,Z 484.181,A -85,B 0,C 180,E1 25883.66,E2 25883.66} C_VEL
LIN {X 0,Y 594.466,Z 572.503,A -85,B 0,C 180,E1 25882.141,E2 25882.141} C_VEL
LIN {X 0,Y 590.322,Z 666.993,A -85,B 0,C 180,E1 25880.633,E2 25880.633} C_VEL
LIN {X 0,Y 586.772,Z 779.948,A -85,B 0,C 180,E1 25878.966,E2 25878.966} C_VEL
LIN {X 0,Y 583.946,Z 891.518,A -85,B 0,C 180,E1 25877.402,E2 25877.402} C_VEL
LIN {X 0,Y 582.072,Z 921.841,A -85,B 0,C 180,E1 25876.833,E2 25876.833} C_VEL
LIN {X 0,Y 580.163,Z 946.001,A -85,B 0,C 180,E1 25876.246,E2 25876.246} C_VEL
LIN {X 0,Y 578.067,Z 969.426,A -85,B 0,C 180,E1 25875.552,E2 25875.552} C_VEL
LIN {X 0,Y 575.255,Z 997.876,A -85,B 0,C 180,E1 25874.535,E2 25874.535} C_VEL
LIN {X 0,Y 572.387,Z 1023.64,A -85,B 0,C 180,E1 25873.417,E2 25873.417} C_VEL
LIN {X 0,Y 569.87,Z 1044.546,A -85,B 0,C 180,E1 25872.38,E2 25872.38} C_VEL
LIN {X 0,Y 567.252,Z 1064.817,A -85,B 0,C 180,E1 25871.242,E2 25871.242} C_VEL
LIN {X 0,Y 564.778,Z 1082.912,A -85,B 0,C 180,E1 25870.109,E2 25870.109} C_VEL
LIN {X 0,Y 562.363,Z 1099.734,A -85,B 0,C 180,E1 25868.95,E2 25868.95} C_VEL
LIN {X 0,Y 559.923,Z 1116.171,A -85,B 0,C 180,E1 25867.712,E2 25867.712} C_VEL
LIN {X 0,Y 557.346,Z 1133.189,A -85,B 0,C 180,E1 25866.3,E2 25866.3} C_VEL
LIN {X 0,Y 555.338,Z 1146.022,A -85,B 0,C 180,E1 25865.117,E2 25865.117} C_VEL
LIN {X 0,Y 552.457,Z 1160.992,A -85,B 0,C 180,E1 25863.45,E2 25863.45} C_VEL
LIN {X 0,Y 549.384,Z 1176.664,A -85,B 0,C 180,E1 25861.489,E2 25861.489} C_VEL
LIN {X 0,Y 546.825,Z 1190.368,A -85,B 0,C 180,E1 25859.584,E2 25859.584} C_VEL
LIN {X 0,Y 544.264,Z 1204.869,A -85,B 0,C 180,E1 25857.341,E2 25857.341} C_VEL
LIN {X 0,Y 541.634,Z 1220.694,A -85,B 0,C 180,E1 25854.542,E2 25854.542} C_VEL
LIN {X 0,Y 539.905,Z 1232.327,A -85,B 0,C 180,E1 25852.181,E2 25852.181} C_VEL
LIN {X 0,Y 538.613,Z 1242.437,A -85,B 0,C 180,E1 25849.86,E2 25849.86} C_VEL
LIN {X 0,Y 537.432,Z 1253.314,A -85,B 0,C 180,E1 25846.983,E2 25846.983} C_VEL
LIN {X 0,Y 536.662,Z 1261.836,A -85,B 0,C 180,E1 25844.237,E2 25844.237} C_VEL
LIN {X 0,Y 536.311,Z 1267.8,A -85,B 0,C 180,E1 25841.943,E2 25841.943} C_VEL
LIN {X 0,Y 536.048,Z 1272.702,A -85,B 0,C 180,E1 25839.664,E2 25839.664} C_VEL
LIN {X 0,Y 535.963,Z 1276.526,A -85,B 0,C 180,E1 25837.396,E2 25837.396} C_VEL
LIN {X 0,Y 535.921,Z 1279.549,A -85,B 0,C 180,E1 25834.923,E2 25834.923} C_VEL
LIN {X 0,Y 535.911,Z 1281.577,A -85,B 0,C 180,E1 25832.031,E2 25832.031} C_VEL
LIN {X 0,Y 535.865,Z 1281.872,A -85,B 0,C 180,E1 25829.358,E2 25829.358} C_VEL
LIN {X 0,Y 535.909,Z 1281.082,A -85,B 0,C 180,E1 25827.112,E2 25827.112} C_VEL
LIN {X 0,Y 535.925,Z 1279.207,A -85,B 0,C 180,E1 25824.755,E2 25824.755} C_VEL
LIN {X 0,Y 535.96,Z 1276.205,A -85,B 0,C 180,E1 25822.388,E2 25822.388} C_VEL
LIN {X 0,Y 536.094,Z 1272.055,A -85,B 0,C 180,E1 25819.997,E2 25819.997} C_VEL
LIN {X 0,Y 536.46,Z 1265.471,A -85,B 0,C 180,E1 25817.076,E2 25817.076} C_VEL
LIN {X 0,Y 537.052,Z 1257.354,A -85,B 0,C 180,E1 25814.272,E2 25814.272} C_VEL
LIN {X 0,Y 537.834,Z 1249.295,A -85,B 0,C 180,E1 25811.913,E2 25811.913} C_VEL
LIN {X 0,Y 538.966,Z 1239.688,A -85,B 0,C 180,E1 25809.474,E2 25809.474} C_VEL
LIN {X 0,Y 540.852,Z 1225.974,A -85,B 0,C 180,E1 25806.488,E2 25806.488} C_VEL
LIN {X 0,Y 542.816,Z 1213.356,A -85,B 0,C 180,E1 25804.116,E2 25804.116} C_VEL
LIN {X 0,Y 544.95,Z 1200.667,A -85,B 0,C 180,E1 25801.985,E2 25801.985} C_VEL
LIN {X 0,Y 547.768,Z 1185.45,A -85,B 0,C 180,E1 25799.702,E2 25799.702} C_VEL
LIN {X 0,Y 551.377,Z 1166.53,A -85,B 0,C 180,E1 25797.218,E2 25797.218} C_VEL
LIN {X 0,Y 554.453,Z 1150.784,A -85,B 0,C 180,E1 25795.385,E2 25795.385} C_VEL
LIN {X 0,Y 557.022,Z 1136.188,A -85,B 0,C 180,E1 25793.93,E2 25793.93} C_VEL
LIN {X 0,Y 560.111,Z 1118.099,A -85,B 0,C 180,E1 25792.309,E2 25792.309} C_VEL
LIN {X 0,Y 563.274,Z 1099.505,A -85,B 0,C 180,E1 25790.807,E2 25790.807} C_VEL
LIN {X 0,Y 567.28,Z 1075.457,A -85,B 0,C 180,E1 25789.075,E2 25789.075} C_VEL
LIN {X 0,Y 570.991,Z 1051.764,A -85,B 0,C 180,E1 25787.609,E2 25787.609} C_VEL
LIN {X 0,Y 573.953,Z 1031.813,A -85,B 0,C 180,E1 25786.518,E2 25786.518} C_VEL
LIN {X 0,Y 576.769,Z 1011.629,A -85,B 0,C 180,E1 25785.544,E2 25785.544} C_VEL
LIN {X 0,Y 579.512,Z 990.607,A -85,B 0,C 180,E1 25784.66,E2 25784.66} C_VEL
LIN {X 0,Y 582.586,Z 964.686,A -85,B 0,C 180,E1 25783.735,E2 25783.735} C_VEL
LIN {X 0,Y 585.193,Z 938.01,A -85,B 0,C 180,E1 25782.987,E2 25782.987} C_VEL
LIN {X 0,Y 586.985,Z 916.549,A -85,B 0,C 180,E1 25782.509,E2 25782.509} C_VEL
LIN {X 0,Y 588.355,Z 894.495,A -85,B 0,C 180,E1 25782.121,E2 25782.121} C_VEL
LIN {X 0,Y 596.133,Z 670.115,A -85,B 0,C 180,E1 25778.837,E2 25778.837} C_VEL
LIN {X 0,Y 603.549,Z 483.918,A -85,B 0,C 180,E1 25776.024,E2 25776.024} C_VEL
LIN {X 0,Y 598.652,Z 454.586,A -85,B 0,C 180,E1 25774.777,E2 25774.777} C_VEL
LIN {X 0,Y 585.204,Z 433.859,A -85,B 0,C 180,E1 25772.504,E2 25772.504} C_VEL
LIN {X 0,Y 570.418,Z 412.677,A -85,B 0,C 180,E1 25769.799,E2 25769.799} C_VEL
LIN {X 0,Y 567.75,Z 408.526,A -85,B 0,C 180,E1 25769.199,E2 25769.199} C_VEL
LIN {X 0,Y 559.948,Z 393.961,A -85,B 0,C 180,E1 25766.514,E2 25766.514} C_VEL
LIN {X 0,Y 554.087,Z 383.576,A -85,B 0,C 180,E1 25764.409,E2 25764.409} C_VEL
LIN {X 0,Y 551.399,Z 378.819,A -85,B 0,C 180,E1 25763.399,E2 25763.399} C_VEL
LIN {X 0,Y 549.092,Z 374.576,A -85,B 0,C 180,E1 25762.483,E2 25762.483} C_VEL
LIN {X 0,Y 546.785,Z 370.466,A -85,B 0,C 180,E1 25761.566,E2 25761.566} C_VEL
LIN {X 0,Y 544.009,Z 365.718,A -85,B 0,C 180,E1 25760.44,E2 25760.44} C_VEL
LIN {X 0,Y 540.999,Z 360.758,A -85,B 0,C 180,E1 25759.207,E2 25759.207} C_VEL
LIN {X 0,Y 540.338,Z 359.379,A -85,B 0,C 180,E1 25758.895,E2 25758.895} C_VEL
LIN {X 0,Y 538.224,Z 356.495,A -85,B 0,C 180,E1 25758.074,E2 25758.074} C_VEL
LIN {X 0,Y 537.65,Z 354.458,A -85,B 0,C 180,E1 25757.562,E2 25757.562} C_VEL
LIN {X 0,Y 537.599,Z 354.253,A -85,B 0,C 180,E1 25754.212,E2 25754.212} C_VEL
LIN {X 0,Y 537.622,Z 354.254,A -85,B 0,C 180,E1 25750.827,E2 25750.827} C_VEL
LIN {X 0,Y 537.617,Z 354.259,A -85,B 0,C 180,E1 25747.373,E2 25747.373} C_VEL
LIN {X 0,Y 537.596,Z 354.26,A -85,B 0,C 180,E1 25743.946,E2 25743.946} C_VEL
LIN {X 0,Y 537.626,Z 354.252,A -85,B 0,C 180,E1 25740.533,E2 25740.533} C_VEL
LIN {X 0,Y 537.605,Z 354.26,A -85,B 0,C 180,E1 25737.122,E2 25737.122} C_VEL
LIN {X 0,Y 537.594,Z 354.263,A -85,B 0,C 180,E1 25733.7,E2 25733.7} C_VEL
LIN {X 0,Y 537.628,Z 354.262,A -85,B 0,C 180,E1 25730.364,E2 25730.364} C_VEL
LIN {X 0,Y 537.592,Z 354.263,A -85,B 0,C 180,E1 25726.994,E2 25726.994} C_VEL
LIN {X 0,Y 537.601,Z 354.257,A -85,B 0,C 180,E1 25723.578,E2 25723.578} C_VEL
LIN {X 0,Y 537.625,Z 354.254,A -85,B 0,C 180,E1 25720.215,E2 25720.215} C_VEL
LIN {X 0,Y 537.58,Z 354.254,A -85,B 0,C 180,E1 25716.892,E2 25716.892} C_VEL
LIN {X 0,Y 537.614,Z 354.253,A -85,B 0,C 180,E1 25713.489,E2 25713.489} C_VEL
LIN {X 0,Y 537.601,Z 354.251,A -85,B 0,C 180,E1 25710.225,E2 25710.225} C_VEL
LIN {X 0,Y 537.581,Z 354.259,A -85,B 0,C 180,E1 25706.822,E2 25706.822} C_VEL
LIN {X 0,Y 537.627,Z 354.253,A -85,B 0,C 180,E1 25703.459,E2 25703.459} C_VEL
LIN {X 0,Y 537.578,Z 354.263,A -85,B 0,C 180,E1 25700.189,E2 25700.189} C_VEL
LIN {X 0,Y 537.592,Z 354.264,A -85,B 0,C 180,E1 25696.807,E2 25696.807} C_VEL
LIN {X 0,Y 537.614,Z 354.261,A -85,B 0,C 180,E1 25693.483,E2 25693.483} C_VEL
LIN {X 0,Y 537.569,Z 354.269,A -85,B 0,C 180,E1 25690.197,E2 25690.197} C_VEL
LIN {X 0,Y 537.621,Z 354.266,A -85,B 0,C 180,E1 25686.895,E2 25686.895} C_VEL
LIN {X 0,Y 537.575,Z 354.267,A -85,B 0,C 180,E1 25683.562,E2 25683.562} C_VEL
LIN {X 0,Y 537.571,Z 354.26,A -85,B 0,C 180,E1 25680.127,E2 25680.127} C_VEL
LIN {X 0,Y 537.605,Z 354.255,A -85,B 0,C 180,E1 25676.988,E2 25676.988} C_VEL
LIN {X 0,Y 537.559,Z 354.254,A -85,B 0,C 180,E1 25673.689,E2 25673.689} C_VEL
LIN {X 0,Y 537.621,Z 354.251,A -85,B 0,C 180,E1 25670.466,E2 25670.466} C_VEL
LIN {X 0,Y 537.559,Z 354.263,A -85,B 0,C 180,E1 25667.202,E2 25667.202} C_VEL
LIN {X 0,Y 537.571,Z 354.271,A -85,B 0,C 180,E1 25663.773,E2 25663.773} C_VEL
LIN {X 0,Y 537.582,Z 354.264,A -85,B 0,C 180,E1 25660.611,E2 25660.611} C_VEL
LIN {X 0,Y 537.546,Z 354.262,A -85,B 0,C 180,E1 25657.267,E2 25657.267} C_VEL
LIN {X 0,Y 537.609,Z 354.262,A -85,B 0,C 180,E1 25654.053,E2 25654.053} C_VEL
LIN {X 0,Y 537.543,Z 354.266,A -85,B 0,C 180,E1 25650.853,E2 25650.853} C_VEL
LIN {X 0,Y 537.564,Z 354.261,A -85,B 0,C 180,E1 25650.4,E2 25650.4} C_VEL
LIN {X 0,Y 537.868,Z 355.225,A -85,B 0,C 180,E1 25649.834,E2 25649.834} C_VEL
LIN {X 0,Y 538.751,Z 358.229,A -85,B 0,C 180,E1 25649.215,E2 25649.215} C_VEL
LIN {X 0,Y 540.598,Z 364.019,A -85,B 0,C 180,E1 25648.497,E2 25648.497} C_VEL
LIN {X 0,Y 544.452,Z 373.565,A -85,B 0,C 180,E1 25647.472,E2 25647.472} C_VEL
LIN {X 0,Y 544.831,Z 374.273,A -85,B 0,C 180,E1 25647.381,E2 25647.381} C_VEL
LIN {X 0,Y 548.153,Z 378.689,A -85,B 0,C 180,E1 25646.654,E2 25646.654} C_VEL
LIN {X 0,Y 549.854,Z 380.673,A -85,B 0,C 180,E1 25646.299,E2 25646.299} C_VEL
LIN {X 0,Y 553.627,Z 385.247,A -85,B 0,C 180,E1 25645.53,E2 25645.53} C_VEL
LIN {X 0,Y 559.963,Z 393.04,A -85,B 0,C 180,E1 25644.289,E2 25644.289} C_VEL
LIN {X 0,Y 568.705,Z 404.032,A -85,B 0,C 180,E1 25642.649,E2 25642.649} C_VEL
LIN {X 0,Y 580.272,Z 418.935,A -85,B 0,C 180,E1 25640.629,E2 25640.629} C_VEL
LIN {X 0,Y 591.559,Z 434.268,A -85,B 0,C 180,E1 25638.792,E2 25638.792} C_VEL
LIN {X 0,Y 596.216,Z 441.011,A -85,B 0,C 180,E1 25638.064,E2 25638.064} C_VEL
LIN {X 0,Y 588.103,Z 636.659,A -85,B 0,C 180,E1 25635.118,E2 25635.118} C_VEL
LIN {X 0,Y 583.333,Z 763.176,A -85,B 0,C 180,E1 25633.245,E2 25633.245} C_VEL
LIN {X 0,Y 581.492,Z 790.933,A -85,B 0,C 180,E1 25632.691,E2 25632.691} C_VEL
LIN {X 0,Y 579.182,Z 815.987,A -85,B 0,C 180,E1 25632.013,E2 25632.013} C_VEL
LIN {X 0,Y 576.915,Z 836.653,A -85,B 0,C 180,E1 25631.328,E2 25631.328} C_VEL
LIN {X 0,Y 574.338,Z 857.122,A -85,B 0,C 180,E1 25630.526,E2 25630.526} C_VEL
LIN {X 0,Y 571.388,Z 878.063,A -85,B 0,C 180,E1 25629.567,E2 25629.567} C_VEL
LIN {X 0,Y 567.406,Z 902.951,A -85,B 0,C 180,E1 25628.232,E2 25628.232} C_VEL
LIN {X 0,Y 563.694,Z 923.784,A -85,B 0,C 180,E1 25626.921,E2 25626.921} C_VEL
LIN {X 0,Y 559.994,Z 943.208,A -85,B 0,C 180,E1 25625.529,E2 25625.529} C_VEL
LIN {X 0,Y 555.722,Z 964.527,A -85,B 0,C 180,E1 25623.787,E2 25623.787} C_VEL
LIN {X 0,Y 551.287,Z 985.256,A -85,B 0,C 180,E1 25621.822,E2 25621.822} C_VEL
LIN {X 0,Y 547.24,Z 1003.823,A -85,B 0,C 180,E1 25619.797,E2 25619.797} C_VEL
LIN {X 0,Y 542.906,Z 1023.605,A -85,B 0,C 180,E1 25617.318,E2 25617.318} C_VEL
LIN {X 0,Y 539.348,Z 1041.374,A -85,B 0,C 180,E1 25614.842,E2 25614.842} C_VEL
LIN {X 0,Y 536.304,Z 1057.736,A -85,B 0,C 180,E1 25612.234,E2 25612.234} C_VEL
LIN {X 0,Y 533.819,Z 1072.068,A -85,B 0,C 180,E1 25609.603,E2 25609.603} C_VEL
LIN {X 0,Y 531.694,Z 1086.04,A -85,B 0,C 180,E1 25606.654,E2 25606.654} C_VEL
LIN {X 0,Y 530.197,Z 1097.614,A -85,B 0,C 180,E1 25603.798,E2 25603.798} C_VEL
LIN {X 0,Y 529.162,Z 1106.949,A -85,B 0,C 180,E1 25601.068,E2 25601.068} C_VEL
LIN {X 0,Y 528.518,Z 1115.064,A -85,B 0,C 180,E1 25598.217,E2 25598.217} C_VEL
LIN {X 0,Y 528.146,Z 1121.71,A -85,B 0,C 180,E1 25595.318,E2 25595.318} C_VEL
LIN {X 0,Y 527.949,Z 1126.254,A -85,B 0,C 180,E1 25592.668,E2 25592.668} C_VEL
LIN {X 0,Y 527.927,Z 1129.655,A -85,B 0,C 180,E1 25589.876,E2 25589.876} C_VEL
LIN {X 0,Y 527.871,Z 1131.43,A -85,B 0,C 180,E1 25587.284,E2 25587.284} C_VEL
LIN {X 0,Y 527.89,Z 1131.947,A -85,B 0,C 180,E1 25584.61,E2 25584.61} C_VEL
LIN {X 0,Y 527.922,Z 1131.055,A -85,B 0,C 180,E1 25581.867,E2 25581.867} C_VEL
LIN {X 0,Y 527.938,Z 1128.642,A -85,B 0,C 180,E1 25579.079,E2 25579.079} C_VEL
LIN {X 0,Y 528.015,Z 1124.972,A -85,B 0,C 180,E1 25576.389,E2 25576.389} C_VEL
LIN {X 0,Y 528.205,Z 1119.781,A -85,B 0,C 180,E1 25573.688,E2 25573.688} C_VEL
LIN {X 0,Y 528.68,Z 1113.001,A -85,B 0,C 180,E1 25570.902,E2 25570.902} C_VEL
LIN {X 0,Y 529.453,Z 1104.364,A -85,B 0,C 180,E1 25568.034,E2 25568.034} C_VEL
LIN {X 0,Y 530.613,Z 1094.066,A -85,B 0,C 180,E1 25565.19,E2 25565.19} C_VEL
LIN {X 0,Y 532.343,Z 1081.514,A -85,B 0,C 180,E1 25562.25,E2 25562.25} C_VEL
LIN {X 0,Y 534.467,Z 1068.296,A -85,B 0,C 180,E1 25559.571,E2 25559.571} C_VEL
LIN {X 0,Y 537.272,Z 1052.491,A -85,B 0,C 180,E1 25556.799,E2 25556.799} C_VEL
LIN {X 0,Y 540.448,Z 1035.852,A -85,B 0,C 180,E1 25554.266,E2 25554.266} C_VEL
LIN {X 0,Y 546.218,Z 1009.421,A -85,B 0,C 180,E1 25550.73,E2 25550.73} C_VEL
LIN {X 0,Y 550.283,Z 991.655,A -85,B 0,C 180,E1 25548.683,E2 25548.683} C_VEL
LIN {X 0,Y 553.818,Z 975.619,A -85,B 0,C 180,E1 25547.063,E2 25547.063} C_VEL
LIN {X 0,Y 557.101,Z 960.031,A -85,B 0,C 180,E1 25545.659,E2 25545.659} C_VEL
LIN {X 0,Y 560.561,Z 942.661,A -85,B 0,C 180,E1 25544.269,E2 25544.269} C_VEL
LIN {X 0,Y 564.709,Z 920.027,A -85,B 0,C 180,E1 25542.694,E2 25542.694} C_VEL
LIN {X 0,Y 567.895,Z 900.344,A -85,B 0,C 180,E1 25541.523,E2 25541.523} C_VEL
LIN {X 0,Y 570.593,Z 881.725,A -85,B 0,C 180,E1 25540.552,E2 25540.552} C_VEL
LIN {X 0,Y 573.045,Z 862.53,A -85,B 0,C 180,E1 25539.682,E2 25539.682} C_VEL
LIN {X 0,Y 575.534,Z 840.086,A -85,B 0,C 180,E1 25538.816,E2 25538.816} C_VEL
LIN {X 0,Y 577.823,Z 813.485,A -85,B 0,C 180,E1 25537.994,E2 25537.994} C_VEL
LIN {X 0,Y 579.228,Z 792.043,A -85,B 0,C 180,E1 25537.473,E2 25537.473} C_VEL
LIN {X 0,Y 580.248,Z 770.493,A -85,B 0,C 180,E1 25537.066,E2 25537.066} C_VEL
LIN {X 0,Y 585.332,Z 640.144,A -85,B 0,C 180,E1 25535.09,E2 25535.09} C_VEL
LIN {X 0,Y 590.385,Z 549.434,A -85,B 0,C 180,E1 25533.6,E2 25533.6} C_VEL
LIN {X 0,Y 596.307,Z 472.306,A -85,B 0,C 180,E1 25532.239,E2 25532.239} C_VEL
LIN {X 0,Y 599.257,Z 440.816,A -85,B 0,C 180,E1 25531.646,E2 25531.646} C_VEL
LIN {X 0,Y 596.287,Z 432.8,A -85,B 0,C 180,E1 25530.462,E2 25530.462} C_VEL
LIN {X 0,Y 594.927,Z 428.462,A -85,B 0,C 180,E1 25529.527,E2 25529.527} C_VEL
LIN {X 0,Y 594.719,Z 427.674,A -85,B 0,C 180,E1 25529.262,E2 25529.262} C_VEL
LIN {X 0,Y 593.273,Z 432.547,A -85,B 0,C 180,E1 25528.332,E2 25528.332} C_VEL
LIN {X 0,Y 592.788,Z 439.025,A -85,B 0,C 180,E1 25527.433,E2 25527.433} C_VEL
LIN {X 0,Y 593.636,Z 450.216,A -85,B 0,C 180,E1 25526.188,E2 25526.188} C_VEL
LIN {X 0,Y 594.457,Z 454.561,A -85,B 0,C 180,E1 25525.732,E2 25525.732} C_VEL
LIN {X 0,Y 594.903,Z 476.904,A -85,B 0,C 180,E1 25524.718,E2 25524.718} C_VEL
LIN {X 0,Y 595.529,Z 486.412,A -85,B 0,C 180,E1 25524.281,E2 25524.281} C_VEL
LIN {X 0,Y 590.062,Z 563.122,A -85,B 0,C 180,E1 25522.915,E2 25522.915} C_VEL
LIN {X 0,Y 585.514,Z 648.981,A -85,B 0,C 180,E1 25521.482,E2 25521.482} C_VEL
LIN {X 0,Y 581.176,Z 765.16,A -85,B 0,C 180,E1 25519.699,E2 25519.699} C_VEL
LIN {X 0,Y 577.624,Z 890.992,A -85,B 0,C 180,E1 25517.894,E2 25517.894} C_VEL
LIN {X 0,Y 575.657,Z 920.451,A -85,B 0,C 180,E1 25517.324,E2 25517.324} C_VEL
LIN {X 0,Y 573.637,Z 944.713,A -85,B 0,C 180,E1 25516.727,E2 25516.727} C_VEL
LIN {X 0,Y 571.194,Z 970.703,A -85,B 0,C 180,E1 25515.944,E2 25515.944} C_VEL
LIN {X 0,Y 568.076,Z 999.873,A -85,B 0,C 180,E1 25514.859,E2 25514.859} C_VEL
LIN {X 0,Y 565.517,Z 1022.218,A -85,B 0,C 180,E1 25513.875,E2 25513.875} C_VEL
LIN {X 0,Y 562.964,Z 1042.487,A -85,B 0,C 180,E1 25512.863,E2 25512.863} C_VEL
LIN {X 0,Y 560.298,Z 1062.649,A -85,B 0,C 180,E1 25511.731,E2 25511.731} C_VEL
LIN {X 0,Y 557.517,Z 1082.428,A -85,B 0,C 180,E1 25510.483,E2 25510.483} C_VEL
LIN {X 0,Y 554.197,Z 1104.93,A -85,B 0,C 180,E1 25508.892,E2 25508.892} C_VEL
LIN {X 0,Y 550.485,Z 1128.75,A -85,B 0,C 180,E1 25506.957,E2 25506.957} C_VEL
LIN {X 0,Y 547.681,Z 1146.256,A -85,B 0,C 180,E1 25505.361,E2 25505.361} C_VEL
LIN {X 0,Y 545.179,Z 1161.574,A -85,B 0,C 180,E1 25503.816,E2 25503.816} C_VEL
LIN {X 0,Y 542.975,Z 1173.283,A -85,B 0,C 180,E1 25502.403,E2 25502.403} C_VEL
LIN {X 0,Y 539.826,Z 1188.826,A -85,B 0,C 180,E1 25500.252,E2 25500.252} C_VEL
LIN {X 0,Y 537.287,Z 1202.066,A -85,B 0,C 180,E1 25498.209,E2 25498.209} C_VEL
LIN {X 0,Y 534.96,Z 1215.255,A -85,B 0,C 180,E1 25495.936,E2 25495.936} C_VEL
LIN {X 0,Y 532.533,Z 1230.197,A -85,B 0,C 180,E1 25492.988,E2 25492.988} C_VEL
LIN {X 0,Y 530.999,Z 1241.059,A -85,B 0,C 180,E1 25490.502,E2 25490.502} C_VEL
LIN {X 0,Y 529.889,Z 1250.104,A -85,B 0,C 180,E1 25488.14,E2 25488.14} C_VEL
LIN {X 0,Y 529.011,Z 1259.062,A -85,B 0,C 180,E1 25485.429,E2 25485.429} C_VEL
LIN {X 0,Y 528.382,Z 1267.044,A -85,B 0,C 180,E1 25482.455,E2 25482.455} C_VEL
LIN {X 0,Y 528.101,Z 1272.286,A -85,B 0,C 180,E1 25480.031,E2 25480.031} C_VEL
LIN {X 0,Y 527.963,Z 1276.204,A -85,B 0,C 180,E1 25477.727,E2 25477.727} C_VEL
LIN {X 0,Y 527.928,Z 1279.092,A -85,B 0,C 180,E1 25475.434,E2 25475.434} C_VEL
LIN {X 0,Y 527.91,Z 1280.946,A -85,B 0,C 180,E1 25473.149,E2 25473.149} C_VEL
LIN {X 0,Y 527.874,Z 1281.804,A -85,B 0,C 180,E1 25470.977,E2 25470.977} C_VEL
LIN {X 0,Y 527.888,Z 1281.758,A -85,B 0,C 180,E1 25468.806,E2 25468.806} C_VEL
LIN {X 0,Y 527.911,Z 1280.81,A -85,B 0,C 180,E1 25466.634,E2 25466.634} C_VEL
LIN {X 0,Y 527.936,Z 1278.75,A -85,B 0,C 180,E1 25464.239,E2 25464.239} C_VEL
LIN {X 0,Y 528.036,Z 1274.907,A -85,B 0,C 180,E1 25461.397,E2 25461.397} C_VEL
LIN {X 0,Y 528.253,Z 1269.325,A -85,B 0,C 180,E1 25458.536,E2 25458.536} C_VEL
LIN {X 0,Y 528.616,Z 1263.348,A -85,B 0,C 180,E1 25456.1,E2 25456.1} C_VEL
LIN {X 0,Y 529.182,Z 1256.856,A -85,B 0,C 180,E1 25453.874,E2 25453.874} C_VEL
LIN {X 0,Y 530.016,Z 1248.889,A -85,B 0,C 180,E1 25451.522,E2 25451.522} C_VEL
LIN {X 0,Y 531.312,Z 1238.769,A -85,B 0,C 180,E1 25448.934,E2 25448.934} C_VEL
LIN {X 0,Y 533.301,Z 1225.282,A -85,B 0,C 180,E1 25445.993,E2 25445.993} C_VEL
LIN {X 0,Y 535.289,Z 1213.318,A -85,B 0,C 180,E1 25443.717,E2 25443.717} C_VEL
LIN {X 0,Y 537.547,Z 1200.665,A -85,B 0,C 180,E1 25441.564,E2 25441.564} C_VEL
LIN {X 0,Y 540.473,Z 1185.741,A -85,B 0,C 180,E1 25439.296,E2 25439.296} C_VEL
LIN {X 0,Y 544.148,Z 1167.33,A -85,B 0,C 180,E1 25436.843,E2 25436.843} C_VEL
LIN {X 0,Y 547.164,Z 1150.5,A -85,B 0,C 180,E1 25434.985,E2 25434.985} C_VEL
LIN {X 0,Y 550.237,Z 1133.392,A -85,B 0,C 180,E1 25433.284,E2 25433.284} C_VEL
LIN {X 0,Y 553.398,Z 1115.807,A -85,B 0,C 180,E1 25431.704,E2 25431.704} C_VEL
LIN {X 0,Y 557.254,Z 1094.262,A -85,B 0,C 180,E1 25429.965,E2 25429.965} C_VEL
LIN {X 0,Y 561.404,Z 1070.057,A -85,B 0,C 180,E1 25428.268,E2 25428.268} C_VEL
LIN {X 0,Y 564.544,Z 1050.867,A -85,B 0,C 180,E1 25427.078,E2 25427.078} C_VEL
LIN {X 0,Y 567.648,Z 1030.856,A -85,B 0,C 180,E1 25425.975,E2 25425.975} C_VEL
LIN {X 0,Y 570.733,Z 1009.634,A -85,B 0,C 180,E1 25424.946,E2 25424.946} C_VEL
LIN {X 0,Y 574.153,Z 984.505,A -85,B 0,C 180,E1 25423.901,E2 25423.901} C_VEL
LIN {X 0,Y 577.286,Z 957.664,A -85,B 0,C 180,E1 25422.996,E2 25422.996} C_VEL
LIN {X 0,Y 579.555,Z 935.241,A -85,B 0,C 180,E1 25422.381,E2 25422.381} C_VEL
LIN {X 0,Y 581.39,Z 913.798,A -85,B 0,C 180,E1 25421.91,E2 25421.91} C_VEL
LIN {X 0,Y 582.845,Z 890.167,A -85,B 0,C 180,E1 25421.502,E2 25421.502} C_VEL
LIN {X 0,Y 590.796,Z 671.071,A -85,B 0,C 180,E1 25418.269,E2 25418.269} C_VEL
LIN {X 0,Y 598.607,Z 485.992,A -85,B 0,C 180,E1 25415.446,E2 25415.446} C_VEL
LIN {X 0,Y 594.228,Z 459.589,A -85,B 0,C 180,E1 25414.312,E2 25414.312} C_VEL
LIN {X 0,Y 581.614,Z 440.03,A -85,B 0,C 180,E1 25412.146,E2 25412.146} C_VEL
LIN {X 0,Y 567.191,Z 419.205,A -85,B 0,C 180,E1 25409.462,E2 25409.462} C_VEL
LIN {X 0,Y 558.771,Z 407.308,A -85,B 0,C 180,E1 25407.727,E2 25407.727} C_VEL
LIN {X 0,Y 552.001,Z 394.766,A -85,B 0,C 180,E1 25405.308,E2 25405.308} C_VEL
LIN {X 0,Y 546.323,Z 384.673,A -85,B 0,C 180,E1 25403.172,E2 25403.172} C_VEL
LIN {X 0,Y 543.985,Z 380.473,A -85,B 0,C 180,E1 25402.25,E2 25402.25} C_VEL
LIN {X 0,Y 540.875,Z 375.116,A -85,B 0,C 180,E1 25401.004,E2 25401.004} C_VEL
LIN {X 0,Y 538.458,Z 370.741,A -85,B 0,C 180,E1 25399.979,E2 25399.979} C_VEL
LIN {X 0,Y 536.222,Z 367.032,A -85,B 0,C 180,E1 25399.046,E2 25399.046} C_VEL
LIN {X 0,Y 535.265,Z 365.361,A -85,B 0,C 180,E1 25398.629,E2 25398.629} C_VEL
LIN {X 0,Y 533.114,Z 361.788,A -85,B 0,C 180,E1 25397.689,E2 25397.689} C_VEL
LIN {X 0,Y 532.214,Z 360.18,A -85,B 0,C 180,E1 25397.268,E2 25397.268} C_VEL
LIN {X 0,Y 530.047,Z 356.891,A -85,B 0,C 180,E1 25396.325,E2 25396.325} C_VEL
LIN {X 0,Y 529.691,Z 355.453,A -85,B 0,C 180,E1 25395.953,E2 25395.953} C_VEL
LIN {X 0,Y 529.681,Z 355.237,A -85,B 0,C 180,E1 25392.649,E2 25392.649} C_VEL
LIN {X 0,Y 529.683,Z 355.234,A -85,B 0,C 180,E1 25389.156,E2 25389.156} C_VEL
LIN {X 0,Y 529.655,Z 355.237,A -85,B 0,C 180,E1 25385.81,E2 25385.81} C_VEL
LIN {X 0,Y 529.679,Z 355.236,A -85,B 0,C 180,E1 25382.38,E2 25382.38} C_VEL
LIN {X 0,Y 529.687,Z 355.247,A -85,B 0,C 180,E1 25378.918,E2 25378.918} C_VEL
LIN {X 0,Y 529.652,Z 355.25,A -85,B 0,C 180,E1 25375.452,E2 25375.452} C_VEL
LIN {X 0,Y 529.685,Z 355.253,A -85,B 0,C 180,E1 25372.079,E2 25372.079} C_VEL
LIN {X 0,Y 529.676,Z 355.25,A -85,B 0,C 180,E1 25368.678,E2 25368.678} C_VEL
LIN {X 0,Y 529.647,Z 355.252,A -85,B 0,C 180,E1 25365.346,E2 25365.346} C_VEL
LIN {X 0,Y 529.688,Z 355.243,A -85,B 0,C 180,E1 25361.966,E2 25361.966} C_VEL
LIN {X 0,Y 529.664,Z 355.251,A -85,B 0,C 180,E1 25358.538,E2 25358.538} C_VEL
LIN {X 0,Y 529.647,Z 355.256,A -85,B 0,C 180,E1 25355.103,E2 25355.103} C_VEL
LIN {X 0,Y 529.695,Z 355.252,A -85,B 0,C 180,E1 25351.718,E2 25351.718} C_VEL
LIN {X 0,Y 529.65,Z 355.254,A -85,B 0,C 180,E1 25348.364,E2 25348.364} C_VEL
LIN {X 0,Y 529.642,Z 355.247,A -85,B 0,C 180,E1 25344.828,E2 25344.828} C_VEL
LIN {X 0,Y 529.692,Z 355.242,A -85,B 0,C 180,E1 25341.469,E2 25341.469} C_VEL
LIN {X 0,Y 529.636,Z 355.245,A -85,B 0,C 180,E1 25338.208,E2 25338.208} C_VEL
LIN {X 0,Y 529.653,Z 355.244,A -85,B 0,C 180,E1 25334.761,E2 25334.761} C_VEL
LIN {X 0,Y 529.671,Z 355.24,A -85,B 0,C 180,E1 25331.458,E2 25331.458} C_VEL
LIN {X 0,Y 529.627,Z 355.248,A -85,B 0,C 180,E1 25328.122,E2 25328.122} C_VEL
LIN {X 0,Y 529.675,Z 355.244,A -85,B 0,C 180,E1 25324.757,E2 25324.757} C_VEL
LIN {X 0,Y 529.635,Z 355.251,A -85,B 0,C 180,E1 25321.529,E2 25321.529} C_VEL
LIN {X 0,Y 529.63,Z 355.256,A -85,B 0,C 180,E1 25318.04,E2 25318.04} C_VEL
LIN {X 0,Y 529.679,Z 355.251,A -85,B 0,C 180,E1 25314.769,E2 25314.769} C_VEL
LIN {X 0,Y 529.62,Z 355.254,A -85,B 0,C 180,E1 25311.485,E2 25311.485} C_VEL
LIN {X 0,Y 529.656,Z 355.244,A -85,B 0,C 180,E1 25308.149,E2 25308.149} C_VEL
LIN {X 0,Y 529.624,Z 355.247,A -85,B 0,C 180,E1 25304.989,E2 25304.989} C_VEL
LIN {X 0,Y 529.618,Z 355.258,A -85,B 0,C 180,E1 25301.522,E2 25301.522} C_VEL
LIN {X 0,Y 529.684,Z 355.247,A -85,B 0,C 180,E1 25298.139,E2 25298.139} C_VEL
LIN {X 0,Y 529.609,Z 355.25,A -85,B 0,C 180,E1 25294.874,E2 25294.874} C_VEL
LIN {X 0,Y 529.627,Z 355.277,A -85,B 0,C 180,E1 25291.406,E2 25291.406} C_VEL
LIN {X 0,Y 529.69,Z 355.789,A -85,B 0,C 180,E1 25291.028,E2 25291.028} C_VEL
LIN {X 0,Y 530.41,Z 357.879,A -85,B 0,C 180,E1 25290.702,E2 25290.702} C_VEL
LIN {X 0,Y 532.613,Z 360.522,A -85,B 0,C 180,E1 25290.161,E2 25290.161} C_VEL
LIN {X 0,Y 534.707,Z 362.061,A -85,B 0,C 180,E1 25289.692,E2 25289.692} C_VEL
LIN {X 0,Y 536.785,Z 365.573,A -85,B 0,C 180,E1 25289.173,E2 25289.173} C_VEL
LIN {X 0,Y 540.086,Z 368.551,A -85,B 0,C 180,E1 25288.446,E2 25288.446} C_VEL
LIN {X 0,Y 542.934,Z 372.538,A -85,B 0,C 180,E1 25287.784,E2 25287.784} C_VEL
LIN {X 0,Y 544.831,Z 374.273,A -85,B 0,C 180,E1 25287.381,E2 25287.381} C_VEL
LIN {X 0,Y 547.738,Z 381.043,A -85,B 0,C 180,E1 25286.659,E2 25286.659} C_VEL
LIN {X 0,Y 552.287,Z 393.058,A -85,B 0,C 180,E1 25285.539,E2 25285.539} C_VEL
LIN {X 0,Y 555.12,Z 397.451,A -85,B 0,C 180,E1 25284.953,E2 25284.953} C_VEL
LIN {X 0,Y 555.59,Z 397.945,A -85,B 0,C 180,E1 25284.863,E2 25284.863} C_VEL
LIN {X 0,Y 570.497,Z 417.057,A -85,B 0,C 180,E1 25282.065,E2 25282.065} C_VEL
LIN {X 0,Y 584.345,Z 435.402,A -85,B 0,C 180,E1 25279.707,E2 25279.707} C_VEL
LIN {X 0,Y 591.122,Z 445.258,A -85,B 0,C 180,E1 25278.613,E2 25278.613} C_VEL
LIN {X 0,Y 582.376,Z 647.828,A -85,B 0,C 180,E1 25275.543,E2 25275.543} C_VEL
LIN {X 0,Y 577.742,Z 764.62,A -85,B 0,C 180,E1 25273.796,E2 25273.796} C_VEL
LIN {X 0,Y 575.751,Z 793.144,A -85,B 0,C 180,E1 25273.215,E2 25273.215} C_VEL
LIN {X 0,Y 573.485,Z 816.978,A -85,B 0,C 180,E1 25272.563,E2 25272.563} C_VEL
LIN {X 0,Y 571.128,Z 837.776,A -85,B 0,C 180,E1 25271.868,E2 25271.868} C_VEL
LIN {X 0,Y 568.392,Z 858.764,A -85,B 0,C 180,E1 25271.037,E2 25271.037} C_VEL
LIN {X 0,Y 564.869,Z 882.853,A -85,B 0,C 180,E1 25269.916,E2 25269.916} C_VEL
LIN {X 0,Y 560.695,Z 907.211,A -85,B 0,C 180,E1 25268.557,E2 25268.557} C_VEL
LIN {X 0,Y 557.275,Z 925.783,A -85,B 0,C 180,E1 25267.365,E2 25267.365} C_VEL
LIN {X 0,Y 553.796,Z 943.451,A -85,B 0,C 180,E1 25266.088,E2 25266.088} C_VEL
LIN {X 0,Y 549.983,Z 961.818,A -85,B 0,C 180,E1 25264.593,E2 25264.593} C_VEL
LIN {X 0,Y 545.171,Z 983.869,A -85,B 0,C 180,E1 25262.537,E2 25262.537} C_VEL
LIN {X 0,Y 540.64,Z 1003.82,A -85,B 0,C 180,E1 25260.372,E2 25260.372} C_VEL
LIN {X 0,Y 536.34,Z 1022.559,A -85,B 0,C 180,E1 25258.022,E2 25258.022} C_VEL
LIN {X 0,Y 532.423,Z 1039.816,A -85,B 0,C 180,E1 25255.532,E2 25255.532} C_VEL
LIN {X 0,Y 529.133,Z 1056.318,A -85,B 0,C 180,E1 25252.887,E2 25252.887} C_VEL
LIN {X 0,Y 526.401,Z 1070.975,A -85,B 0,C 180,E1 25250.2,E2 25250.2} C_VEL
LIN {X 0,Y 524.328,Z 1083.69,A -85,B 0,C 180,E1 25247.541,E2 25247.541} C_VEL
LIN {X 0,Y 522.602,Z 1095.719,A -85,B 0,C 180,E1 25244.602,E2 25244.602} C_VEL
LIN {X 0,Y 521.414,Z 1105.687,A -85,B 0,C 180,E1 25241.715,E2 25241.715} C_VEL
LIN {X 0,Y 520.651,Z 1114.22,A -85,B 0,C 180,E1 25238.761,E2 25238.761} C_VEL
LIN {X 0,Y 520.172,Z 1121.156,A -85,B 0,C 180,E1 25235.758,E2 25235.758} C_VEL
LIN {X 0,Y 519.961,Z 1125.896,A -85,B 0,C 180,E1 25233.027,E2 25233.027} C_VEL
LIN {X 0,Y 519.933,Z 1129.352,A -85,B 0,C 180,E1 25230.292,E2 25230.292} C_VEL
LIN {X 0,Y 519.885,Z 1131.316,A -85,B 0,C 180,E1 25227.548,E2 25227.548} C_VEL
LIN {X 0,Y 519.896,Z 1131.977,A -85,B 0,C 180,E1 25224.789,E2 25224.789} C_VEL
LIN {X 0,Y 519.922,Z 1131.096,A -85,B 0,C 180,E1 25221.907,E2 25221.907} C_VEL
LIN {X 0,Y 519.939,Z 1128.748,A -85,B 0,C 180,E1 25219.082,E2 25219.082} C_VEL
LIN {X 0,Y 520.025,Z 1125.045,A -85,B 0,C 180,E1 25216.304,E2 25216.304} C_VEL
LIN {X 0,Y 520.231,Z 1119.882,A -85,B 0,C 180,E1 25213.561,E2 25213.561} C_VEL
LIN {X 0,Y 520.756,Z 1112.831,A -85,B 0,C 180,E1 25210.622,E2 25210.622} C_VEL
LIN {X 0,Y 521.582,Z 1104.184,A -85,B 0,C 180,E1 25207.712,E2 25207.712} C_VEL
LIN {X 0,Y 522.833,Z 1093.854,A -85,B 0,C 180,E1 25204.827,E2 25204.827} C_VEL
LIN {X 0,Y 524.602,Z 1081.827,A -85,B 0,C 180,E1 25201.966,E2 25201.966} C_VEL
LIN {X 0,Y 526.859,Z 1068.606,A -85,B 0,C 180,E1 25199.239,E2 25199.239} C_VEL
LIN {X 0,Y 529.808,Z 1052.832,A -85,B 0,C 180,E1 25196.429,E2 25196.429} C_VEL
LIN {X 0,Y 535.261,Z 1028.045,A -85,B 0,C 180,E1 25192.594,E2 25192.594} C_VEL
LIN {X 0,Y 539.461,Z 1010.923,A -85,B 0,C 180,E1 25190.29,E2 25190.29} C_VEL
LIN {X 0,Y 543.659,Z 993.04,A -85,B 0,C 180,E1 25188.22,E2 25188.22} C_VEL
LIN {X 0,Y 547.203,Z 977.483,A -85,B 0,C 180,E1 25186.635,E2 25186.635} C_VEL
LIN {X 0,Y 550.593,Z 961.886,A -85,B 0,C 180,E1 25185.217,E2 25185.217} C_VEL
LIN {X 0,Y 554.16,Z 944.51,A -85,B 0,C 180,E1 25183.813,E2 25183.813} C_VEL
LIN {X 0,Y 558.563,Z 921.079,A -85,B 0,C 180,E1 25182.175,E2 25182.175} C_VEL
LIN {X 0,Y 561.714,Z 902.192,A -85,B 0,C 180,E1 25181.043,E2 25181.043} C_VEL
LIN {X 0,Y 564.491,Z 883.593,A -85,B 0,C 180,E1 25180.063,E2 25180.063} C_VEL
LIN {X 0,Y 567.013,Z 864.406,A -85,B 0,C 180,E1 25179.186,E2 25179.186} C_VEL
LIN {X 0,Y 569.799,Z 840.036,A -85,B 0,C 180,E1 25178.241,E2 25178.241} C_VEL
LIN {X 0,Y 571.968,Z 814.611,A -85,B 0,C 180,E1 25177.463,E2 25177.463} C_VEL
LIN {X 0,Y 573.379,Z 793.659,A -85,B 0,C 180,E1 25176.949,E2 25176.949} C_VEL
LIN {X 0,Y 574.455,Z 771.485,A -85,B 0,C 180,E1 25176.527,E2 25176.527} C_VEL
LIN {X 0,Y 579.563,Z 651.906,A -85,B 0,C 180,E1 25174.675,E2 25174.675} C_VEL
LIN {X 0,Y 584.616,Z 568.196,A -85,B 0,C 180,E1 25173.271,E2 25173.271} C_VEL
LIN {X 0,Y 591.027,Z 490.523,A -85,B 0,C 180,E1 25171.876,E2 25171.876} C_VEL
LIN {X 0,Y 595.775,Z 445.221,A -85,B 0,C 180,E1 25170.999,E2 25170.999} C_VEL
LIN {X 0,Y 593.916,Z 439.065,A -85,B 0,C 180,E1 25169.999,E2 25169.999} C_VEL
LIN {X 0,Y 593.238,Z 436.042,A -85,B 0,C 180,E1 25169.327,E2 25169.327} C_VEL
LIN {X 0,Y 591.599,Z 441.39,A -85,B 0,C 180,E1 25168.403,E2 25168.403} C_VEL
LIN {X 0,Y 590.873,Z 448.552,A -85,B 0,C 180,E1 25167.515,E2 25167.515} C_VEL
LIN {X 0,Y 591.502,Z 459.317,A -85,B 0,C 180,E1 25166.313,E2 25166.313} C_VEL
LIN {X 0,Y 591.323,Z 481.164,A -85,B 0,C 180,E1 25165.28,E2 25165.28} C_VEL
LIN {X 0,Y 591.572,Z 488.738,A -85,B 0,C 180,E1 25164.927,E2 25164.927} C_VEL
LIN {X 0,Y 585.111,Z 567.228,A -85,B 0,C 180,E1 25163.48,E2 25163.48} C_VEL
LIN {X 0,Y 579.942,Z 654.024,A -85,B 0,C 180,E1 25161.991,E2 25161.991} C_VEL
LIN {X 0,Y 575.33,Z 764.304,A -85,B 0,C 180,E1 25160.253,E2 25160.253} C_VEL
LIN {X 0,Y 571.408,Z 889.231,A -85,B 0,C 180,E1 25158.418,E2 25158.418} C_VEL
LIN {X 0,Y 569.353,Z 918.567,A -85,B 0,C 180,E1 25157.839,E2 25157.839} C_VEL
LIN {X 0,Y 567.231,Z 942.766,A -85,B 0,C 180,E1 25157.24,E2 25157.24} C_VEL
LIN {X 0,Y 564.559,Z 969.883,A -85,B 0,C 180,E1 25156.416,E2 25156.416} C_VEL
LIN {X 0,Y 561.422,Z 997.932,A -85,B 0,C 180,E1 25155.359,E2 25155.359} C_VEL
LIN {X 0,Y 558.818,Z 1019.722,A -85,B 0,C 180,E1 25154.395,E2 25154.395} C_VEL
LIN {X 0,Y 556.044,Z 1040.898,A -85,B 0,C 180,E1 25153.333,E2 25153.333} C_VEL
LIN {X 0,Y 553.26,Z 1061.179,A -85,B 0,C 180,E1 25152.185,E2 25152.185} C_VEL
LIN {X 0,Y 550.146,Z 1082.781,A -85,B 0,C 180,E1 25150.808,E2 25150.808} C_VEL
LIN {X 0,Y 546.227,Z 1108.17,A -85,B 0,C 180,E1 25148.953,E2 25148.953} C_VEL
LIN {X 0,Y 543.222,Z 1126.865,A -85,B 0,C 180,E1 25147.402,E2 25147.402} C_VEL
LIN {X 0,Y 540.488,Z 1143.536,A -85,B 0,C 180,E1 25145.875,E2 25145.875} C_VEL
LIN {X 0,Y 537.649,Z 1160.389,A -85,B 0,C 180,E1 25144.169,E2 25144.169} C_VEL
LIN {X 0,Y 535.031,Z 1175.879,A -85,B 0,C 180,E1 25142.435,E2 25142.435} C_VEL
LIN {X 0,Y 533.26,Z 1185.731,A -85,B 0,C 180,E1 25141.165,E2 25141.165} C_VEL
LIN {X 0,Y 530.32,Z 1200.022,A -85,B 0,C 180,E1 25138.973,E2 25138.973} C_VEL
LIN {X 0,Y 527.881,Z 1212.714,A -85,B 0,C 180,E1 25136.795,E2 25136.795} C_VEL
LIN {X 0,Y 525.765,Z 1224.701,A -85,B 0,C 180,E1 25134.493,E2 25134.493} C_VEL
LIN {X 0,Y 523.667,Z 1238.001,A -85,B 0,C 180,E1 25131.583,E2 25131.583} C_VEL
LIN {X 0,Y 522.213,Z 1248.484,A -85,B 0,C 180,E1 25128.88,E2 25128.88} C_VEL
LIN {X 0,Y 521.315,Z 1256.597,A -85,B 0,C 180,E1 25126.461,E2 25126.461} C_VEL
LIN {X 0,Y 520.669,Z 1263.349,A -85,B 0,C 180,E1 25124.116,E2 25124.116} C_VEL
LIN {X 0,Y 520.304,Z 1269.07,A -85,B 0,C 180,E1 25121.753,E2 25121.753} C_VEL
LIN {X 0,Y 520.033,Z 1274.541,A -85,B 0,C 180,E1 25118.96,E2 25118.96} C_VEL
LIN {X 0,Y 519.946,Z 1278.521,A -85,B 0,C 180,E1 25116.071,E2 25116.071} C_VEL
LIN {X 0,Y 519.912,Z 1280.742,A -85,B 0,C 180,E1 25113.528,E2 25113.528} C_VEL
LIN {X 0,Y 519.896,Z 1281.735,A -85,B 0,C 180,E1 25111.322,E2 25111.322} C_VEL
LIN {X 0,Y 519.869,Z 1281.826,A -85,B 0,C 180,E1 25109.118,E2 25109.118} C_VEL
LIN {X 0,Y 519.91,Z 1281.014,A -85,B 0,C 180,E1 25106.913,E2 25106.913} C_VEL
LIN {X 0,Y 519.928,Z 1279.202,A -85,B 0,C 180,E1 25104.593,E2 25104.593} C_VEL
LIN {X 0,Y 519.965,Z 1276.359,A -85,B 0,C 180,E1 25102.264,E2 25102.264} C_VEL
LIN {X 0,Y 520.128,Z 1272.282,A -85,B 0,C 180,E1 25099.813,E2 25099.813} C_VEL
LIN {X 0,Y 520.467,Z 1266.526,A -85,B 0,C 180,E1 25097.124,E2 25097.124} C_VEL
LIN {X 0,Y 521.149,Z 1258.268,A -85,B 0,C 180,E1 25094.076,E2 25094.076} C_VEL
LIN {X 0,Y 522.033,Z 1250.102,A -85,B 0,C 180,E1 25091.577,E2 25091.577} C_VEL
LIN {X 0,Y 523.223,Z 1241.061,A -85,B 0,C 180,E1 25089.179,E2 25089.179} C_VEL
LIN {X 0,Y 524.862,Z 1230.199,A -85,B 0,C 180,E1 25086.656,E2 25086.656} C_VEL
LIN {X 0,Y 527.439,Z 1215.258,A -85,B 0,C 180,E1 25083.666,E2 25083.666} C_VEL
LIN {X 0,Y 529.899,Z 1202.064,A -85,B 0,C 180,E1 25081.362,E2 25081.362} C_VEL
LIN {X 0,Y 532.592,Z 1188.822,A -85,B 0,C 180,E1 25079.293,E2 25079.293} C_VEL
LIN {X 0,Y 534.358,Z 1179.684,A -85,B 0,C 180,E1 25078.025,E2 25078.025} C_VEL
LIN {X 0,Y 537.45,Z 1163.031,A -85,B 0,C 180,E1 25076.01,E2 25076.01} C_VEL
LIN {X 0,Y 540.597,Z 1146.334,A -85,B 0,C 180,E1 25074.185,E2 25074.185} C_VEL
LIN {X 0,Y 544.386,Z 1126.425,A -85,B 0,C 180,E1 25072.227,E2 25072.227} C_VEL
LIN {X 0,Y 548.668,Z 1103.303,A -85,B 0,C 180,E1 25070.234,E2 25070.234} C_VEL
LIN {X 0,Y 552.173,Z 1084.065,A -85,B 0,C 180,E1 25068.766,E2 25068.766} C_VEL
LIN {X 0,Y 555.52,Z 1065.242,A -85,B 0,C 180,E1 25067.479,E2 25067.479} C_VEL
LIN {X 0,Y 558.837,Z 1045.787,A -85,B 0,C 180,E1 25066.291,E2 25066.291} C_VEL
LIN {X 0,Y 562.278,Z 1024.494,A -85,B 0,C 180,E1 25065.141,E2 25065.141} C_VEL
LIN {X 0,Y 566.306,Z 997.11,A -85,B 0,C 180,E1 25063.879,E2 25063.879} C_VEL
LIN {X 0,Y 569.349,Z 974.017,A -85,B 0,C 180,E1 25062.992,E2 25062.992} C_VEL
LIN {X 0,Y 571.91,Z 952.42,A -85,B 0,C 180,E1 25062.297,E2 25062.297} C_VEL
LIN {X 0,Y 574.215,Z 930.064,A -85,B 0,C 180,E1 25061.707,E2 25061.707} C_VEL
LIN {X 0,Y 576.544,Z 902.146,A -85,B 0,C 180,E1 25061.136,E2 25061.136} C_VEL
LIN {X 0,Y 578.523,Z 853.867,A -85,B 0,C 180,E1 25060.401,E2 25060.401} C_VEL
LIN {X 0,Y 586.342,Z 652.733,A -85,B 0,C 180,E1 25057.397,E2 25057.397} C_VEL
LIN {X 0,Y 593.633,Z 487.657,A -85,B 0,C 180,E1 25054.844,E2 25054.844} C_VEL
LIN {X 0,Y 589.822,Z 464.514,A -85,B 0,C 180,E1 25053.835,E2 25053.835} C_VEL
LIN {X 0,Y 577.807,Z 445.848,A -85,B 0,C 180,E1 25051.74,E2 25051.74} C_VEL
LIN {X 0,Y 563.951,Z 425.725,A -85,B 0,C 180,E1 25049.123,E2 25049.123} C_VEL
LIN {X 0,Y 552.933,Z 410.381,A -85,B 0,C 180,E1 25046.849,E2 25046.849} C_VEL
LIN {X 0,Y 549.388,Z 405.192,A -85,B 0,C 180,E1 25046.016,E2 25046.016} C_VEL
LIN {X 0,Y 542.393,Z 392.223,A -85,B 0,C 180,E1 25043.35,E2 25043.35} C_VEL
LIN {X 0,Y 536.118,Z 381.422,A -85,B 0,C 180,E1 25040.869,E2 25040.869} C_VEL
LIN {X 0,Y 533.386,Z 376.672,A -85,B 0,C 180,E1 25039.72,E2 25039.72} C_VEL
LIN {X 0,Y 530.491,Z 371.645,A -85,B 0,C 180,E1 25038.461,E2 25038.461} C_VEL
LIN {X 0,Y 528.316,Z 367.871,A -85,B 0,C 180,E1 25037.473,E2 25037.473} C_VEL
LIN {X 0,Y 527.163,Z 366.168,A -85,B 0,C 180,E1 25036.984,E2 25036.984} C_VEL
LIN {X 0,Y 525.135,Z 362.631,A -85,B 0,C 180,E1 25036.027,E2 25036.027} C_VEL
LIN {X 0,Y 524.222,Z 361.116,A -85,B 0,C 180,E1 25035.601,E2 25035.601} C_VEL
LIN {X 0,Y 522.152,Z 357.931,A -85,B 0,C 180,E1 25034.642,E2 25034.642} C_VEL
LIN {X 0,Y 521.741,Z 356.383,A -85,B 0,C 180,E1 25034.138,E2 25034.138} C_VEL
LIN {X 0,Y 521.744,Z 356.233,A -85,B 0,C 180,E1 25030.713,E2 25030.713} C_VEL
LIN {X 0,Y 521.755,Z 356.239,A -85,B 0,C 180,E1 25027.156,E2 25027.156} C_VEL
LIN {X 0,Y 521.716,Z 356.242,A -85,B 0,C 180,E1 25023.736,E2 25023.736} C_VEL
LIN {X 0,Y 521.742,Z 356.236,A -85,B 0,C 180,E1 25020.22,E2 25020.22} C_VEL
LIN {X 0,Y 521.746,Z 356.236,A -85,B 0,C 180,E1 25016.704,E2 25016.704} C_VEL
LIN {X 0,Y 521.715,Z 356.238,A -85,B 0,C 180,E1 25013.286,E2 25013.286} C_VEL
LIN {X 0,Y 521.732,Z 356.24,A -85,B 0,C 180,E1 25009.845,E2 25009.845} C_VEL
LIN {X 0,Y 521.751,Z 356.24,A -85,B 0,C 180,E1 25006.366,E2 25006.366} C_VEL
LIN {X 0,Y 521.709,Z 356.23,A -85,B 0,C 180,E1 25002.948,E2 25002.948} C_VEL
LIN {X 0,Y 521.722,Z 356.232,A -85,B 0,C 180,E1 24999.468,E2 24999.468} C_VEL
LIN {X 0,Y 521.749,Z 356.227,A -85,B 0,C 180,E1 24996.081,E2 24996.081} C_VEL
LIN {X 0,Y 521.703,Z 356.24,A -85,B 0,C 180,E1 24992.738,E2 24992.738} C_VEL
LIN {X 0,Y 521.736,Z 356.237,A -85,B 0,C 180,E1 24989.351,E2 24989.351} C_VEL
LIN {X 0,Y 521.732,Z 356.24,A -85,B 0,C 180,E1 24985.971,E2 24985.971} C_VEL
LIN {X 0,Y 521.698,Z 356.245,A -85,B 0,C 180,E1 24982.51,E2 24982.51} C_VEL
LIN {X 0,Y 521.746,Z 356.241,A -85,B 0,C 180,E1 24979.194,E2 24979.194} C_VEL
LIN {X 0,Y 521.716,Z 356.243,A -85,B 0,C 180,E1 24975.789,E2 24975.789} C_VEL
LIN {X 0,Y 521.696,Z 356.239,A -85,B 0,C 180,E1 24972.426,E2 24972.426} C_VEL
LIN {X 0,Y 521.757,Z 356.23,A -85,B 0,C 180,E1 24969.086,E2 24969.086} C_VEL
LIN {X 0,Y 521.691,Z 356.235,A -85,B 0,C 180,E1 24965.772,E2 24965.772} C_VEL
LIN {X 0,Y 521.699,Z 356.233,A -85,B 0,C 180,E1 24962.304,E2 24962.304} C_VEL
LIN {X 0,Y 521.72,Z 356.228,A -85,B 0,C 180,E1 24959.13,E2 24959.13} C_VEL
LIN {X 0,Y 521.683,Z 356.237,A -85,B 0,C 180,E1 24955.732,E2 24955.732} C_VEL
LIN {X 0,Y 521.738,Z 356.235,A -85,B 0,C 180,E1 24952.419,E2 24952.419} C_VEL
LIN {X 0,Y 521.691,Z 356.247,A -85,B 0,C 180,E1 24949.108,E2 24949.108} C_VEL
LIN {X 0,Y 521.683,Z 356.239,A -85,B 0,C 180,E1 24945.679,E2 24945.679} C_VEL
LIN {X 0,Y 521.721,Z 356.233,A -85,B 0,C 180,E1 24942.507,E2 24942.507} C_VEL
LIN {X 0,Y 521.67,Z 356.244,A -85,B 0,C 180,E1 24939.154,E2 24939.154} C_VEL
LIN {X 0,Y 521.716,Z 356.241,A -85,B 0,C 180,E1 24935.83,E2 24935.83} C_VEL
LIN {X 0,Y 521.681,Z 356.34,A -85,B 0,C 180,E1 24932.856,E2 24932.856} C_VEL
LIN {X 0,Y 522.006,Z 357.695,A -85,B 0,C 180,E1 24932.511,E2 24932.511} C_VEL
LIN {X 0,Y 523.817,Z 360.702,A -85,B 0,C 180,E1 24931.996,E2 24931.996} C_VEL
LIN {X 0,Y 526.925,Z 363.205,A -85,B 0,C 180,E1 24931.25,E2 24931.25} C_VEL
LIN {X 0,Y 529.063,Z 366.722,A -85,B 0,C 180,E1 24930.68,E2 24930.68} C_VEL
LIN {X 0,Y 532.069,Z 369.448,A -85,B 0,C 180,E1 24929.973,E2 24929.973} C_VEL
LIN {X 0,Y 534.808,Z 373.367,A -85,B 0,C 180,E1 24929.304,E2 24929.304} C_VEL
LIN {X 0,Y 537.445,Z 375.803,A -85,B 0,C 180,E1 24928.721,E2 24928.721} C_VEL
LIN {X 0,Y 540.768,Z 380.088,A -85,B 0,C 180,E1 24927.96,E2 24927.96} C_VEL
LIN {X 0,Y 542.53,Z 382.07,A -85,B 0,C 180,E1 24927.571,E2 24927.571} C_VEL
LIN {X 0,Y 547.365,Z 388.17,A -85,B 0,C 180,E1 24926.518,E2 24926.518} C_VEL
LIN {X 0,Y 552.889,Z 394.836,A -85,B 0,C 180,E1 24925.389,E2 24925.389} C_VEL
LIN {X 0,Y 555.59,Z 397.945,A -85,B 0,C 180,E1 24924.863,E2 24924.863} C_VEL
LIN {X 0,Y 558.124,Z 401.599,A -85,B 0,C 180,E1 24924.36,E2 24924.36} C_VEL
LIN {X 0,Y 560.954,Z 408.908,A -85,B 0,C 180,E1 24923.719,E2 24923.719} C_VEL
